	Status();
	
	xResetInterno := FALSE;
	// faz depois dos status o reset automatico do axis
	IF stMotor.Sa.xCmdFwd AND stMotor.Sa.sStatusConexao = 'Parado' AND stHoraAgora.wMilliseconds < 500 THEN
		xResetInterno := TRUE;
	END_IF


END_IF



LeParametros();


xFirstScan := false;

ACTION ControlaACCDEC:

//Pra aparecer na IHM
stMotor.Config.inversor.xtemSuavidadeRampa := TRUE;
stMotor.Config.inversor.xtemACC := TRUE;
stMotor.Config.inversor.xtemDEC := TRUE;

//Pra nao dar exceção
IF stMotor.Config.inversor.SuavidadeRampa < 1 THEN
	stMotor.Config.inversor.SuavidadeRampa := 1;
END_IF
IF stMotor.Config.inversor.SuavidadeRampa > 2 THEN
	stMotor.Config.inversor.SuavidadeRampa := 2;
END_IF

IF stMotor.Config.inversor.ACC < 0.000001 THEN
	stMotor.Config.inversor.ACC := 1;
END_IF

IF stMotor.Config.inversor.DEC < 0.000001 THEN
	stMotor.Config.inversor.DEC := 1;
END_IF

//calculos de verdade
IF xCalcula THEN
	rAux := (stMotor.Sa.iVelocidade*6*stMotor.Config.inversor.SuavidadeRampa)/stMotor.Config.inversor.ACC;
	iAceleracaoCalculada := REAL_TO_UDINT(rAux);
	
	rAux := (stMotor.Sa.iVelocidade*6*stMotor.Config.inversor.SuavidadeRampa)/stMotor.Config.inversor.DEC;
	iDesaceleracaoCalculada := REAL_TO_UDINT(rAux);
	
	rAux := ((stMotor.Sa.iVelocidade*6*stMotor.Config.inversor.SuavidadeRampa)/(stMotor.Config.inversor.ACC*stMotor.Config.inversor.ACC))*((-100.01*stMotor.Config.inversor.SuavidadeRampa)+202.02);
	iJerkCalculado := REAL_TO_UDINT(rAux);
END_IF

//joga nos blocos que precisa
ExAxMvVelo.Acceleration := iAceleracaoCalculada;
ExAxMvVelo.Deceleration := iDesaceleracaoCalculada;
fbMC_Halt.Deceleration := iDesaceleracaoCalculada;


ExAxMvVelo.Jerk := iJerkCalculado;
fbMC_Halt.Jerk := (iJerkCalculado);
ExAxStop.Jerk := (iJerkCalculado);
END_ACTION

ACTION LeParametros:






CASE iEstadoLeCorrente OF
	0: 
		tonEsperaInicio(IN:= TRUE, PT:= T#10S, Q=> , ET=> );
		IF tonEsperaInicio.q THEN
			iEstadoLeCorrente := 1;
		END_IF

	1:

		// tem que no primeiro ciclo jogar uma real nele pra ele conseguir ler depois, nao faz seentido mas vai entender a beckhoffs
		fbReadCorrenteDePico.Execute := TRUE;
		fbReadCorrenteDePico(
			Axis    := AxisREF,
			Idn     := P_0_IDNs + 92,
			Element := 16#40,
			pDstBuf := ADR(rPCorrenteDePico),
			BufLen  := SIZEOF(rPCorrenteDePico),
			Timeout := DEFAULT_ADS_TIMEOUT,
		);
		iEstadoLeCorrente := 2;

		
	2:
		//ai aqui ele so joga um false pra ele nao ficar preso em nada
		fbReadCorrenteDePico(Axis:= AxisREF);
		IF NOT fbReadCorrenteDePico.Busy THEN
			fbReadCorrenteDePico.Execute := FALSE;
			iEstadoLeCorrente := 3;
		END_IF
		
	3:
		//aqui ele faz a logica de verdade e ajeita e fica tudo certo
		IF iAuxCorrenteDePico = 0 AND NOT fbReadCorrenteDePico.Busy THEN
			fbReadCorrenteDePico.Execute := TRUE;
		END_IF
		
		
		fbReadCorrenteDePico(
			Axis    := AxisREF,
			Idn     := P_0_IDNs + 92,
			Element := 16#40,
			pDstBuf := ADR(iAuxCorrenteDePico),
			BufLen  := SIZEOF(iAuxCorrenteDePico),
			Timeout := DEFAULT_ADS_TIMEOUT,
		 );
		
		
		IF NOT fbReadCorrenteDePico.Busy THEN
			fbReadCorrenteDePico.Execute := FALSE;
			fbReadCorrenteDePico(Axis := AxisREF);
			rPCorrenteDePico := iAuxCorrenteDePico;
			rPCorrenteDePico := rPCorrenteDePico/1000;
		END_IF

		
END_CASE
END_ACTION

ACTION Status:


//Erro

ExAxLeErro(
	Axis:= AxisREF, 
	Enable:= TRUE, 
	Valid=> , 
	Busy=> , 
	Error=> , 
	ErrorID=> , 
	AxisErrorID=> );


fbSoEReadDiagNumber(
	Axis:= AxisREF, 
	NetId:= AxisREF.ADS.NetId, 
	Execute:= NOT fbSoEReadDiagNumber.Busy, 
	Timeout:= , 
	Busy=> , 
	Error=> , 
	AdsErrId=> , 
	SercosErrId=> , 
	DiagNumber=> , 
	Attribute=> );
	
fbMCReadStatus(
	Axis:= AxisREF, 
	Enable:= TRUE, 
	Valid=> , 
	Busy=> , 
	Error=> , 
	ErrorID=> , 
	ErrorStop=> , 
	Disabled=> , 
	Stopping=> , 
	StandStill=> , 
	DiscreteMotion=> , 
	ContinuousMotion=> , 
	SynchronizedMotion=> , 
	Homing=> , 
	ConstantVelocity=> , 
	Accelerating=> , 
	Decelerating=> , 
	Status=> );


stMotor.En.xFalhaInversor :=  fbMCReadStatus.Error OR fbSoEReadDiagNumber.DiagNumber < 53266 OR fbSoEReadDiagNumber.DiagNumber > 53268;


fbSoEReadDiagMsg(
	Axis:= AxisREF, 
	NetId:= AxisREF.ADS.NetId, 
	Execute:=  NOT fbSoEReadDiagMsg.Busy, 
	Timeout:= , 
	Busy=> , 
	Error=> , 
	AdsErrId=> , 
	SercosErrId=> , 
	DiagMessage=> , 
	Attribute=> );
	
tonOnline(IN:= fbSoEReadDiagMsg.AdsErrId = 0, PT:= T#5S, Q=> , ET=> );
stMotor.En.xInversorOnline := tonOnline.q;

	
IF fbSoEReadDiagNumber.DiagNumber < 53266 OR fbSoEReadDiagNumber.DiagNumber > 53268 THEN
	stMotor.Sa.sStatusConexao := 'Falha';
	stMotor.Sa.sUltimoErro := fbSoEReadDiagMsg.DiagMessage.strData;
ELSE
	CASE AxisREF.NcToPlc.AxisState OF
		0 :stMotor.Sa.sStatusConexao := 'Parado';
		1,3 :stMotor.Sa.sStatusConexao := 'Rodando';
		4 :stMotor.Sa.sStatusConexao := 'Acelerando';
		5 :stMotor.Sa.sStatusConexao := 'Desacelerando';
	END_CASE
END_IF

IF NOT stMotor.En.xInversorOnline THEN
	stMotor.Sa.sStatusConexao := 'Offline';
END_IF



//Velo
ExAxVeloReal(
	Axis:= AxisREF, 
	Enable:= TRUE, 
	Valid=> , 
	Busy=> , 
	Error=> , 
	ErrorID=> , 
	ActualVelocity=> );
	
IF ExAxVeloReal.ActualVelocity > 1 THEN	
	stMotor.Sa.rVelocidadeRPM := LREAL_TO_REAL(AxisREF.NcToPlc.ActVelo/6);
ELSE
	stMotor.Sa.rVelocidadeRPM := 0;
END_IF


//Temp
(*
ExAxLeTempMotor(
	Axis:= AxisREF, 
	NetId:= '', 
	Execute:= NOT ExAxLeTempMotor.Busy, 
	Timeout:= , 
	Busy=> , 
	Error=> , 
	AdsErrId=> , 
	SercosErrId=> , 
	MotorTemperature=> , 
	Attribute=> );
*)
raux := iTemperaturaMotor;
stMotor.Sa.rTemperaturaMotor := raux/100;//ExAxLeTempMotor.MotorTemperature;

raux := iTemperaturaInversor;
stMotor.Sa.rTemperaturaInver := raux/100;

//Corrente
raux := iCorrente;

iBufferAbsoluteCurrent[iCurrentIndex] := iCorrente;
iCurrentIndex := iCurrentIndex + 1;
IF iCurrentIndex > 10 THEN
	iCurrentIndex := 0;
END_IF
(*
stMotor.Sa.rCorrente := (((iBufferAbsoluteCurrent[0] + 
					iBufferAbsoluteCurrent[1] + iBufferAbsoluteCurrent[2] +
					iBufferAbsoluteCurrent[3] + iBufferAbsoluteCurrent[4] +
					iBufferAbsoluteCurrent[5] + iBufferAbsoluteCurrent[6] +
					iBufferAbsoluteCurrent[7] + iBufferAbsoluteCurrent[8] +
					iBufferAbsoluteCurrent[9])/100)*rPCorrenteDePico)/100;*)
	
				
filtroCorrente(in:= (((raux)/100)*rPCorrenteDePico)/10, T:= T#500MS, K:= 1, out=> stMotor.Sa.rCorrente );		

IF NOT stMotor.Sa.xLigado THEN
	stMotor.Sa.rCorrente := 0;
END_IF

//Torque

stMotor.Sa.rTorque := AxisREF.NcToPlc.ActTorque;

IF NOT stMotor.Sa.xLigado THEN
	stMotor.Sa.rTorque := 0;
END_IF

//Tensao de entrada

stMotor.Sa.rVoltagemEntrada := 0;


stMotor.LeiturasInversorIHM.sCorrente			:= concat(TO_STRING(F_RetiraCasa(stMotor.Sa.rCorrente, 2)), ' A');
stMotor.LeiturasInversorIHM.sStatusConexao		:= stMotor.Sa.sStatusConexao;
stMotor.LeiturasInversorIHM.sTemperaturaInver	:= 'ND';
stMotor.LeiturasInversorIHM.sTemperaturaMotor	:= 'ND';
stMotor.LeiturasInversorIHM.sTorque				:= concat(TO_STRING(F_RetiraCasa(stMotor.Sa.rTorque, 2)), ' %');
stMotor.LeiturasInversorIHM.sUltimoErro			:= stMotor.Sa.sUltimoErro;
//stMotor.LeiturasInversorIHM.sVelocidadeHz		:= concat(TO_STRING(F_RetiraCasa(stMotor.Sa.rVelocidadeRPM, 2)), ' Hz');
stMotor.LeiturasInversorIHM.sVelocidadeRPM		:= concat(TO_STRING(F_RetiraCasa(stMotor.Sa.rVelocidadeRPM, 2)), ' RPM');
END_ACTION

END_FUNCTION_BLOCK

// POUs/Comunicação/CAN/FB_ComunicacaoCanOpen
//{attribute 'hide_all_locals'}
FUNCTION_BLOCK FB_ComunicacaoCanOpen
VAR_IN_OUT
	stMotor	: st_Partida;
	LinkCan	: ATV320_Can;
	Config	: Config_CAN;
END_VAR
VAR_INPUT

END_VAR
VAR_OUTPUT
	ITH_S	: REAL;	//corrente maxima 
	ACC_S	: REAL;	//rampa de aceleração
	DEC_S	: REAL;	//rampa de desaceleração
END_VAR
VAR

	//Maquina
	Ult2ETA	: WORD;
	Ult1ETA	: WORD;

	iEstadoMaquina : MaquinaCanOpen;

	//Escrita SDO
	SDO_WRITE		: ARRAY[1..4] OF SDO_WRITE;
	ReadData		: ARRAY[0..255] OF BYTE;
	WriteDataCTRL	: ARRAY[0..255] OF BYTE;
	uiControlWord	: INT;

	xForcaNST : BOOL;

	//Leitura e escrita
	SDO_READ		: ARRAY[1..4] OF SDO_READ;
	rtComacaLeitura	: R_TRIG;

	ChegouInformacao	: ARRAY[1..4] OF R_TRIG;
	R_TRIGs				: ARRAY[1..10] OF R_TRIG;

	AuxLeitura	: UINT;
	rAux		: REAL;
	
	xAux : BOOL;
	
	iUltimoErro : UINT;
	rtEntrouEmFalha : R_TRIG;
	xPegaUltimoErro : BOOL;
	rtVoltouOnline : R_TRIG;
	
	rtDesligou : R_TRIG;
	iSeguraAlgunsCiclos : INT;

END_VAR


IF xLicensaValida5154156 THEN	
	
	stMotor.En.xTemInversor := TRUE;
	stMotor.En.xResetBlocoComunicacao := FALSE;
	
	Leituras_SDO();
	TrocaEstadoMaquinaDeEstados();
	AcaoMaquinaDeEstados();
	//EscritaPDO();
	Status();
	Escritas_SDO();
	
	// local bloqueado ou em emergencia
	IF xForcaNST OR stMotor.En.xBloqueado (* OR NOT stMotor.En.xEmergenciaOK *) THEN
		LinkCan.Controlword := 0;
	END_IF
ELSE
	ValidaLicensa();
END_IF

ACTION AcaoMaquinaDeEstados:


CASE iEstadoMaquina OF
	SwitchOnDisabled:
		//fica pulsando o sinal para caso ele demore um pouco pra começar a processar os pacotes, ai ele nao fica preso em NST
		IF stMotor.En.stHoraAgora.wMilliseconds > 500 THEN
			LinkCan.Controlword := 16#0006; // manda acionar o drive
		ELSE
			LinkCan.Controlword := 16#0000; // Se comando 
		END_IF

	ReadyToSwitchOn:
		IF stMotor.Sa.xCmdFwd OR stMotor.Sa.xCmdRev THEN
			LinkCan.Controlword := 16#000F; // manda ligar o drive
		END_IF

	SwitchedOn:
		IF stMotor.Sa.xCmdFwd OR stMotor.Sa.xCmdRev THEN
			LinkCan.Controlword := 16#000F; // manda ligar de vez
		ELSE
			LinkCan.Controlword := 16#0007; // manda voltar e e ficar esperando
		END_IF

	OperationEnabled:
		IF NOT (stMotor.Sa.xCmdFwd OR stMotor.Sa.xCmdRev) THEN
			LinkCan.Controlword := 16#0007; // manda desligar o drive
		END_IF

	QuickStopActive:
		LinkCan.Controlword := 16#0000; // a pincipio nao se cai aqui mas caso aconteca ele volta certo

	fault: // caso mandem ele resetar, ou se a falha for COF(erro na can)
		//Caso a falha seja de can ele tenta fazer o reset automatico,
		// ai ele fica pulsando o reset pra caso ele nao pegue o primeiro pacote de reset
		
		LinkCan.Controlword := 16#0006; // manda acionar o drive
		IF (iUltimoErro = 34 AND stMotor.En.xFalhaInversor) THEN
			IF stMotor.En.stHoraAgora.wMilliseconds > 500 THEN
				LinkCan.Controlword := 16#0080; // comando de reset
				stMotor.En.xResetBlocoComunicacao := TRUE;
			ELSE
				LinkCan.Controlword := 16#0000; // Se comando 
			END_IF
		END_IF

		IF stMotor.Sa.xResetParaInversor THEN
			LinkCan.Controlword := 16#0080; // comando de reset
		END_IF

END_CASE

IF stMotor.Sa.xCmdRev THEN
	LinkCan.TargetVelocity := -stMotor.Sa.iVelocidade;
ELSE
	LinkCan.TargetVelocity := stMotor.Sa.iVelocidade;
END_IF

IF stMotor.Sa.xCmdFwd THEN
	IF stMotor.Sa.xResetParaInversor THEN
		LinkCan.TargetVelocity := stMotor.Sa.iVelocidade - 1;
	END_IF
END_IF
END_ACTION

ACTION EscritaPDO:



(*
rtDesligou(CLK:=NOT stMotor.Sa.xLigado);
IF rtDesligou.q OR  iSeguraAlgunsCiclos > 0 AND iSeguraAlgunsCiclos < 20 THEN
	iSeguraAlgunsCiclos := iSeguraAlgunsCiclos +1;
	rAux := Config.Retentiva.NPR-0.1;
	LinkCan.NC1 := REAL_TO_UINT(rAux*10);
	rAux := Config.Retentiva.ITH-0.1;
	LinkCan.NC2 := REAL_TO_UINT(rAux-0.1*10);
	rAux := Config.Retentiva.NSP-0.1;
	LinkCan.NC3 := REAL_TO_UINT(rAux-0.1*10);
	rAux := Config.Retentiva.NCR-0.1;
	LinkCan.NC4 := REAL_TO_UINT(rAux-0.1*10);
ELSE	
	iSeguraAlgunsCiclos := 0;
	LinkCan.NC1 := REAL_TO_UINT(Config.Retentiva.NPR*10);
	LinkCan.NC2 := REAL_TO_UINT(Config.Retentiva.ITH*10);
	LinkCan.NC3 := REAL_TO_UINT(Config.Retentiva.NSP*10);
	LinkCan.NC4 := REAL_TO_UINT(Config.Retentiva.NCR*10);
END_IF
*)
END_ACTION

ACTION Escritas_SDO:

//Corrente
(*
R_TRIGs[1](CLK := Config.normal.xEscreve_ITH, Q =>);

IF R_TRIGs[1].q THEN
	SDO_WRITE[1].StartWriting := TRUE;
END_IF

uiControlWord := TO_INT(Config.Retentiva.ITH_E * 10);
MEMCPY(destAddr := ADR(WriteDataCTRL), srcAddr := ADR(uiControlWord), n := SIZEOF(WriteDataCTRL));

SDO_WRITE[1]
	(
		ADSNetID := Config.Retentiva.sAdressCAN,
			PortNr := 4096 + Config.Retentiva.wPortNrCAN,
			CO_Index := 16#2042,
			CO_SubIndex := 16#17,
			DataLength := SIZEOF(WORD),
			StartWriting :=,
			WriteData := WriteDataCTRL,
			WriteDataFinished =>,
			Error =>);

R_TRIGs[2](CLK := SDO_WRITE[1].WriteDataFinished, Q =>);

IF R_TRIGs[2].q THEN
	Config.normal.xEscreve_ITH	:= FALSE;
	SDO_WRITE[1].StartWriting	:= FALSE;

	Config.normal.xLe := TRUE;
END_IF
*)
//Aceleração

R_TRIGs[3](CLK := Config.normal.xEscreve_ACC, Q =>);

IF R_TRIGs[3].q THEN
	SDO_WRITE[2].StartWriting := TRUE;
END_IF

uiControlWord := TO_INT(Config.Retentiva.ACC_E * 10);
MEMCPY(destAddr := ADR(WriteDataCTRL), srcAddr := ADR(uiControlWord), n := SIZEOF(WriteDataCTRL));

SDO_WRITE[2]
	(
		ADSNetID := Config.Retentiva.sAdressCAN,
			PortNr := 4096 + Config.Retentiva.wPortNrCAN,
			CO_Index := 16#203C,
			CO_SubIndex := 16#2,
			DataLength := SIZEOF(WORD),
			StartWriting :=,
			WriteData := WriteDataCTRL,
			WriteDataFinished =>,
			Error =>);

R_TRIGs[4](CLK := SDO_WRITE[2].WriteDataFinished, Q =>);

IF R_TRIGs[4].q THEN
	SDO_WRITE[2].StartWriting	:= FALSE;
	Config.normal.xEscreve_ACC	:= FALSE;

	Config.normal.xLe := TRUE;
END_IF

//Desaceleração

R_TRIGs[5](CLK := Config.normal.xEscreve_DEC, Q =>);

IF R_TRIGs[5].q THEN
	SDO_WRITE[3].StartWriting := TRUE;
END_IF

uiControlWord := TO_INT(Config.Retentiva.DEC_E * 10);
MEMCPY(destAddr := ADR(WriteDataCTRL), srcAddr := ADR(uiControlWord), n := SIZEOF(WriteDataCTRL));

SDO_WRITE[3]
	(
		ADSNetID := Config.Retentiva.sAdressCAN,
			PortNr := 4096 + Config.Retentiva.wPortNrCAN,
			CO_Index := 16#203C,
			CO_SubIndex := 16#3,
			DataLength := SIZEOF(WORD),
			StartWriting :=,
			WriteData := WriteDataCTRL,
			WriteDataFinished =>,
			Error =>);

R_TRIGs[6](CLK := SDO_WRITE[3].WriteDataFinished, Q =>);

IF R_TRIGs[6].q THEN
	SDO_WRITE[3].StartWriting	:= FALSE;
	Config.normal.xEscreve_DEC	:= FALSE;

	Config.normal.xLe := true;
END_IF
END_ACTION

ACTION Leituras_SDO:

rtComacaLeitura(CLK := Config.Normal.xLe, Q =>);

IF rtComacaLeitura.Q THEN
	//xTerminouLeituras:=FALSE;
END_IF
(*
//////////// ITH
SDO_READ[1]
	(
		StartReading :=,
			CO_Index := 16#2042,
			CO_SubIndex := 16#17,
			DataLength := SIZEOF(UINT),
			PortNr := 4096 + Config.Retentiva.wPortNrCAN,
			ADSNetID := Config.Retentiva.sAdressCAN);

ChegouInformacao[1](CLK := SDO_READ[1].ReadDataAvailable, Q =>);

IF ChegouInformacao[1].q THEN
	Config.Normal.xLe			:= FALSE;
	SDO_READ[2].StartReading	:= TRUE;

	ReadData := SDO_READ[1].ReadData;
	MEMCPY(destAddr := ADR(AuxLeitura), srcAddr := ADR(ReadData), n := SIZEOF(UINT));
	ITH_S					:= UINT_TO_REAL(AuxLeitura) / 10;
	Config.Retentiva.ITH_E	:= ITH_S;
END_IF
*)
//////////// ACC		
SDO_READ[2]
	(
		StartReading := Config.Normal.xLe,
			CO_Index := 16#203C,
			CO_SubIndex := 16#2,
			DataLength := SIZEOF(UINT),
			PortNr := 4096 + Config.Retentiva.wPortNrCAN,
			ADSNetID := Config.Retentiva.sAdressCAN);

ChegouInformacao[2](CLK := SDO_READ[2].ReadDataAvailable, Q =>);

IF ChegouInformacao[2].q THEN
	SDO_READ[2].StartReading	:= FALSE;
	SDO_READ[3].StartReading	:= TRUE;

	ReadData := SDO_READ[2].ReadData;
	MEMCPY(destAddr := ADR(AuxLeitura), srcAddr := ADR(ReadData), n := SIZEOF(UINT));
	ACC_S					:= UINT_TO_REAL(AuxLeitura) / 10;
	Config.Retentiva.ACC_E	:= ACC_S;
END_IF

//////////// DEC		
SDO_READ[3]
	(
		StartReading :=,
			CO_Index := 16#203C,
			CO_SubIndex := 16#3,
			DataLength := SIZEOF(UINT),
			PortNr := 4096 + Config.Retentiva.wPortNrCAN,
			ADSNetID := Config.Retentiva.sAdressCAN);

ChegouInformacao[3](CLK := SDO_READ[3].ReadDataAvailable, Q =>);

IF ChegouInformacao[3].q THEN
	SDO_READ[3].StartReading := FALSE;

	ReadData := SDO_READ[3].ReadData;
	MEMCPY(destAddr := ADR(AuxLeitura), srcAddr := ADR(ReadData), n := SIZEOF(UINT));
	DEC_S					:= UINT_TO_REAL(AuxLeitura) / 10;
	Config.Retentiva.DEC_E	:= DEC_S;
END_IF




SDO_READ[4]
	(
		StartReading :=xPegaUltimoErro,
			CO_Index := 16#2029,
			CO_SubIndex := 16#16,
			DataLength := SIZEOF(UINT),
			PortNr := 4096 + Config.Retentiva.wPortNrCAN,
			ADSNetID := Config.Retentiva.sAdressCAN);

ChegouInformacao[4](CLK := SDO_READ[4].ReadDataAvailable, Q =>);

IF ChegouInformacao[4].q THEN
	xPegaUltimoErro := FALSE;
	ReadData := SDO_READ[4].ReadData;
	MEMCPY(destAddr := ADR(iUltimoErro), srcAddr := ADR(ReadData), n := SIZEOF(UINT));
END_IF
END_ACTION

ACTION Status:

// manda status de online e falha
stMotor.En.xFalhaInversor := iEstadoMaquina = Fault;

//IF  THEN
	IF LinkCan.NodeState <> 31 THEN
		stMotor.En.xInversorOnline :=
			 (LinkCan.NodeState <> 2); // Nao sei se é o melhor jeito, mas o 2 é o unico que fala especificamente de o inversor nao ter sido encontrado
										// nao o 31 pq se nao ele buga e fica dando reset pra sempre nos inversor	
	END_IF
//END_IF
								
rAux							:= LinkCan.NM2;
stMotor.Sa.rCorrente			:= rAux / 10;
stMotor.Sa.rTemperaturaMotor	:= LinkCan.NM3;
rAux							:= LinkCan.NM4;
stMotor.Sa.rTorque				:= rAux/10;

stMotor.Sa.rVelocidadeRPM	:= LinkCan.ControlEffort;
rAux						:= stMotor.Sa.rVelocidadeRPM;
stMotor.Sa.rVelocidadeHZ	:= rAux * 0.016667 * 2;

stMotor.LeiturasInversorIHM.sCorrente			:= concat(TO_STRING(F_RetiraCasa(stMotor.Sa.rCorrente, 2)), ' A');
stMotor.LeiturasInversorIHM.sStatusConexao		:= stMotor.Sa.sStatusConexao;
stMotor.LeiturasInversorIHM.sTemperaturaInver	:= 'ND';
stMotor.LeiturasInversorIHM.sTemperaturaMotor	:= concat(TO_STRING(F_RetiraCasa(stMotor.Sa.rTemperaturaMotor, 2)), ' %');
stMotor.LeiturasInversorIHM.sTorque				:= concat(TO_STRING(F_RetiraCasa(stMotor.Sa.rTorque, 2)), ' %');
stMotor.LeiturasInversorIHM.sUltimoErro			:= stMotor.Sa.sUltimoErro;
stMotor.LeiturasInversorIHM.sVelocidadeHz		:= concat(TO_STRING(F_RetiraCasa(stMotor.Sa.rVelocidadeHZ, 2)), ' Hz');

IF stMotor.Config.xVeloEmMetroPMin THEN
	rAux										:= (stMotor.Sa.rVelocidadeRPM * stMotor.Config.rVeloEmMetroPMin_Conversao) / 1800;	
	stMotor.Sa.rVeloComissionada				:= rAux;
	stMotor.LeiturasInversorIHM.sVelocidadeRPM	:= concat(TO_STRING(F_RetiraCasa(rAux, 2)), ' m/Min');
ELSIF stMotor.Config.xVeloEmPorcentagem THEN
	IF stMotor.Config.rVeloEmPorcentagem_VeloMax < 0.1 THEN
		stMotor.Config.rVeloEmPorcentagem_VeloMax := 1;
	END_IF
	rAux										:= (stMotor.Sa.rVelocidadeRPM * 100) / stMotor.Config.rVeloEmPorcentagem_VeloMax;
	stMotor.Sa.rVeloComissionada				:= rAux;
	stMotor.LeiturasInversorIHM.sVelocidadeRPM	:= concat(TO_STRING(F_RetiraCasa(rAux, 2)), ' %');
ELSE
	stMotor.Sa.rVeloComissionada				:= stMotor.Sa.rVelocidadeRPM;
	stMotor.LeiturasInversorIHM.sVelocidadeRPM := concat(TO_STRING(F_RetiraCasa(stMotor.Sa.rVelocidadeRPM, 2)), ' RPM');
END_IF

stMotor.LeiturasInversorIHM.sVoltagemEntrada := 'ND';

config.Normal.rITH_Lido	:= ITH_S;
config.Normal.rACC_Lido	:= ACC_S;
config.Normal.rDEC_Lido	:= DEC_S;

// 30 é STO
xAux := LinkCan.NM1 = 30;
stMotor.En.xEmergenciaOK := stMotor.En.xEmergenciaOK AND NOT xAux;

CASE LinkCan.NM1 OF
	0:
		IF iUltimoErro = 0 THEN
			stMotor.Sa.sStatusConexao := 'Offline';
		ELSE
			stMotor.Sa.sStatusConexao := '[Autotuning] (TUN)';
		END_IF

	1:
		stMotor.Sa.sStatusConexao := '[Injeção de CC] (DCB)';

	2:
		stMotor.Sa.sStatusConexao := '[Pronto] (RDY)';

	3:
		stMotor.Sa.sStatusConexao := '[Esperando] (NST)';

	4:
		stMotor.Sa.sStatusConexao := '[Rodando] (RUN)';

	5:
		stMotor.Sa.sStatusConexao := '[Acelerando] (ACC)';

	6:
		stMotor.Sa.sStatusConexao := '[Desacelerando] (DEC)';

	7:
		stMotor.Sa.sStatusConexao := '[Limitando Corrente] (CLI)';

	8:
		stMotor.Sa.sStatusConexao := '[Parada Rapida] (FST)';

	11:
		stMotor.Sa.sStatusConexao := '[Sem Tensão de Entrada] (NLP)';

	13:
		stMotor.Sa.sStatusConexao := '[control.stop] (CTL)';

	14:
		stMotor.Sa.sStatusConexao := '[Dec. adapt.] (OBR)';

	15:
		stMotor.Sa.sStatusConexao := '[Output cut] (SOC)';

	17:
		stMotor.Sa.sStatusConexao := '[Undervoltage Warning] (USA)';

	18:
		stMotor.Sa.sStatusConexao := '[TC Mode Active] (TC)';

	19:
		stMotor.Sa.sStatusConexao := '[In autotest] (ST)';

	20:
		stMotor.Sa.sStatusConexao := '[Autotest error] (FA)';

	21:
		stMotor.Sa.sStatusConexao := '[Autotest OK] (OK)';

	22:
		stMotor.Sa.sStatusConexao := '[EEprom test] (EP))';

	23:
		stMotor.Sa.sStatusConexao := '[Falha] (FLT)';

	25:
		stMotor.Sa.sStatusConexao := '[DCP Flashing Mode] (DCP)';

	30:
		stMotor.Sa.sStatusConexao := '[Emergencia Ativa] (STO)';

	35:
		stMotor.Sa.sStatusConexao := '[Salvando Energia] (IDLE)';

	36:
		stMotor.Sa.sStatusConexao := '[Atualizando Firmware] (FWUP)';

	37:
		stMotor.Sa.sStatusConexao := '[AFE Mains Undervoltage ] (URA)';
END_CASE

IF NOT stMotor.En.xInversorOnline THEN
	stMotor.Sa.sStatusConexao := 'Offline';
END_IF

CASE iUltimoErro OF
	0:
		stMotor.Sa.sUltimoErro := 'Carregando';

	2:
		stMotor.Sa.sUltimoErro := '[EEPROM Control] (EEF1)';

	3:
		stMotor.Sa.sUltimoErro := '[Configuração Incorreta] (CFF)';

	4:
		stMotor.Sa.sUltimoErro := '[Configuração Invalida] (CFI)';

	5:
		stMotor.Sa.sUltimoErro := '[Com. ModBus Interrompida] (SLF1)';

	6:
		stMotor.Sa.sUltimoErro := '[Internal Link Error] (ILF)';

	7:
		stMotor.Sa.sUltimoErro := '[Fieldbus Com Interrupt] (CNF)';

	8:
		stMotor.Sa.sUltimoErro := '[Erro Externo] (EPF1)';

	9:
		stMotor.Sa.sUltimoErro := '[Sobrecorrente] (OCF)';

	10:
		stMotor.Sa.sUltimoErro := '[Precharge Capacitor] (CRF1)';

	11:
		stMotor.Sa.sUltimoErro := '[Encoder Feedback Loss] (SPF)';

	12:
		stMotor.Sa.sUltimoErro := '[Load slipping] (ANF)';

	15:
		stMotor.Sa.sUltimoErro := '[Entrada Superaquecendo] (IHF)';

	16:
		stMotor.Sa.sUltimoErro := '[Inversor Superaquecendo] (OHF)';

	17:
		stMotor.Sa.sUltimoErro := '[Motor Sobracarregado] (OLF)';

	18:
		stMotor.Sa.sUltimoErro := '[DC Bus Sobretensão] (OBF)';

	19:
		stMotor.Sa.sUltimoErro := '[Entrada com Sobretensão] (OSF)';

	20:
		stMotor.Sa.sUltimoErro := '[Perda de 1 Fase da Saida] (OPF1)';

	21:
		stMotor.Sa.sUltimoErro := '[Perda de Fase na Entrada] (PHF)';

	22:
		stMotor.Sa.sUltimoErro := '[Entrada em subtensão] (USF)';

	23:
		stMotor.Sa.sUltimoErro := '[Motor em Curto-Circuito] (SCF1)';

	24:
		stMotor.Sa.sUltimoErro := '[Motor Overspeed] (SOF)';

	25:
		stMotor.Sa.sUltimoErro := '[Autotuning Error] (TNF)';

	26:
		stMotor.Sa.sUltimoErro := '[Internal Error 1] (INF1)';

	27:
		stMotor.Sa.sUltimoErro := '[Internal Error 2] (INF2)';

	28:
		stMotor.Sa.sUltimoErro := '[Internal Error 3] (INF3)';

	29:
		stMotor.Sa.sUltimoErro := '[Internal Error 4] (INF4)';

	30:
		stMotor.Sa.sUltimoErro := '[EEPROM Power] (EEF2)';

	32:
		stMotor.Sa.sUltimoErro := '[Curto-Circuito a Terra] (SCF3)';

	33:
		stMotor.Sa.sUltimoErro := '[Falta de Fase na Saida] (OPF2)';

	34:
		stMotor.Sa.sUltimoErro := '[Com. CANopen Interrompida] (COF)';

	35:
		stMotor.Sa.sUltimoErro := '[Brake Control] (BLF)';

	37:
		stMotor.Sa.sUltimoErro := '[Internal Error 7] (INF7)';

	38:
		stMotor.Sa.sUltimoErro := '[Fieldbus Error] (EPF2)';

	40:
		stMotor.Sa.sUltimoErro := '[Internal Error 8] (INF8)';

	41:
		stMotor.Sa.sUltimoErro := '[Brake Feedback] (BRF)';

	42:
		stMotor.Sa.sUltimoErro := '[PC Com. Interruption] (SLF2)';

	43:
		stMotor.Sa.sUltimoErro := '[Encoder Coupling] (ECF)';

	44:
		stMotor.Sa.sUltimoErro := '[Erro na Limitção de Torque] (SSF)';

	45:
		stMotor.Sa.sUltimoErro := '[Com. HMI Interrompido] (SLF3)';

	51:
		stMotor.Sa.sUltimoErro := '[Internal Error 9] (INF9)';

	52:
		stMotor.Sa.sUltimoErro := '[Internal Error 10] (INFA)';

	53:
		stMotor.Sa.sUltimoErro := '[Internal Error 11] (INFB)';

	54:
		stMotor.Sa.sUltimoErro := '[IGBT Superaquecendo] (TJF)';

	55:
		stMotor.Sa.sUltimoErro := '[IGBT em Curto-Circuito] (SCF4)';

	56:
		stMotor.Sa.sUltimoErro := '[Motor em Curto-Circuito] (SCF5)';

	57:
		stMotor.Sa.sUltimoErro := '[Torque timeout] (SRF)';

	58:
		stMotor.Sa.sUltimoErro := '[Out Contact Closed Error] (FCF1)';

	59:
		stMotor.Sa.sUltimoErro := '[Out Contact Opened Error] (FCF2)';

	60:
		stMotor.Sa.sUltimoErro := '[Internal Error 12] (INFC)';

	62:
		stMotor.Sa.sUltimoErro := '[Encoder] (ENF)';

	64:
		stMotor.Sa.sUltimoErro := '[Input Contactor] (LCF)';

	65:
		stMotor.Sa.sUltimoErro := '[DB unit sh. circuit] (BUF)';

	68:
		stMotor.Sa.sUltimoErro := '[Internal Error 6] (INF6)';

	69:
		stMotor.Sa.sUltimoErro := '[Internal Error 14] (INFE)';

	70:
		stMotor.Sa.sUltimoErro := '[Braking Resistor ovld] (BOF)';

	71:
		stMotor.Sa.sUltimoErro := '[Perda AI3 4-20mA] (LFF3)';

	72:
		stMotor.Sa.sUltimoErro := '[Perda AI4 4-20mA] (LFF4)';

	73:
		stMotor.Sa.sUltimoErro := '[Boards Compatibility] (HCF)';

	76:
		stMotor.Sa.sUltimoErro := '[Dynamic Load Error] (DLF)';

	77:
		stMotor.Sa.sUltimoErro := '[Conf Transfer Error] (CFI2)';

	79:
		stMotor.Sa.sUltimoErro := '[Perda AI5 4-20 mA] (LFF5)';

	99:
		stMotor.Sa.sUltimoErro := '[Channel Switch Error] (CSF)';

	100:
		stMotor.Sa.sUltimoErro := '[Process Underload] (ULF)';

	101:
		stMotor.Sa.sUltimoErro := '[Process Overload] (OLC)';

	105:
		stMotor.Sa.sUltimoErro := '[Angle error] (ASF)';

	106:
		stMotor.Sa.sUltimoErro := '[Perda AI1 4-20 mA] (LFF1)';

	107:
		stMotor.Sa.sUltimoErro := '[Safety Function Error] (SAFF)';

	112:
		stMotor.Sa.sUltimoErro := '[AI3 Th Level Error] (TH3F)';

	113:
		stMotor.Sa.sUltimoErro := '[AI3 Thermal Sensor Error] (T3CF)';

	120:
		stMotor.Sa.sUltimoErro := '[AI4 Th Level Error] (TH4F)';

	121:
		stMotor.Sa.sUltimoErro := '[AI4 Thermal Sensor Error] (T4CF)';

	122:
		stMotor.Sa.sUltimoErro := '[AI5 Th Level Error] (TH5F)';

	123:
		stMotor.Sa.sUltimoErro := '[AI5 Thermal Sensor Error] (T5CF)';

	128:
		stMotor.Sa.sUltimoErro := '[Program Loading Error] (PGLF)';

	129:
		stMotor.Sa.sUltimoErro := '[Program Running Error] (PGRF)';

	142:
		stMotor.Sa.sUltimoErro := '[Internal Error 16] (INFG)';

	143:
		stMotor.Sa.sUltimoErro := '[Internal Error 17] (INFH)';

	144:
		stMotor.Sa.sUltimoErro := '[Internal Error 0] (INF0)';

	146:
		stMotor.Sa.sUltimoErro := '[Internal Error 13] (INFD)';

	148:
		stMotor.Sa.sUltimoErro := '[Motor Stall Error] (STF)';

	149:
		stMotor.Sa.sUltimoErro := '[Internal Error 21] (INFL)';

	150:
		stMotor.Sa.sUltimoErro := '[Com. Embd Eth Interrompida] (ETHF)';

	151:
		stMotor.Sa.sUltimoErro := '[Internal Error 15] (INFF)';

	152:
		stMotor.Sa.sUltimoErro := '[Firmware Update Error] (FWER)';

	153:
		stMotor.Sa.sUltimoErro := '[Internal Error 22] (INFM)';

	154:
		stMotor.Sa.sUltimoErro := '[Internal Error 25] (INFP)';

	155:
		stMotor.Sa.sUltimoErro := '[Internal Error 20] (INFK)';

	156:
		stMotor.Sa.sUltimoErro := '[Internal Error 19] (INFJ)';

	157:
		stMotor.Sa.sUltimoErro := '[Internal Error 27] (INFR)';

	158:
		stMotor.Sa.sUltimoErro := '[Internal Error 23] (INFN)';

	159:
		stMotor.Sa.sUltimoErro := '[AFE ShortCircuit error] (SCF6)';

	160:
		stMotor.Sa.sUltimoErro := '[AFE Bus unbalancing ] (OBF2)';

	161:
		stMotor.Sa.sUltimoErro := '[Internal Error 28] (INFS)';

	173:
		stMotor.Sa.sUltimoErro := '[Cabinet Overheat  Error] (CHF)';

	175:
		stMotor.Sa.sUltimoErro := '[Internal Error 31] (INFV)';

	176:
		stMotor.Sa.sUltimoErro := '[Internal Error 29] (INFT)';

	177:
		stMotor.Sa.sUltimoErro := '[Internal Error 30] (INFU)';

	179:
		stMotor.Sa.sUltimoErro := '[AFE IGBT over-heat error] (TJF2)';

	180:
		stMotor.Sa.sUltimoErro := '[AFE contactor feedback error] (CRF3)';

	181:
		stMotor.Sa.sUltimoErro := '[Pre-settings Transfer Error] (CFI3)';

	182:
		stMotor.Sa.sUltimoErro := '[Circuit Breaker Error] (CBF)';

	184:
		stMotor.Sa.sUltimoErro := '[DB unit op. circuit] (BUFO)';

	185:
		stMotor.Sa.sUltimoErro := '[Inversor Sobrecarregado] (TLOF)';

	186:
		stMotor.Sa.sUltimoErro := '[MultiDrive Link Error] (MDLF)';

	187:
		stMotor.Sa.sUltimoErro := '[AI1 Th Level Error] (TH1F)';

	188:
		stMotor.Sa.sUltimoErro := '[AI1 Thermal Sensor Error] (T1CF)';

	189:
		stMotor.Sa.sUltimoErro := '[Backlash Error] (BSQF)';

	190:
		stMotor.Sa.sUltimoErro := '[M/S Device Error] (MSDF)';

	194:
		stMotor.Sa.sUltimoErro := '[Encoder Th Level Error] (THEF)';

	195:
		stMotor.Sa.sUltimoErro := '[Encoder Th Sensor Error] (TECF)';

	196:
		stMotor.Sa.sUltimoErro := '[Sem Configuração] (CFI4)';

	200:
		stMotor.Sa.sUltimoErro := '[FDR 1 Error] (FDR1)';

	201:
		stMotor.Sa.sUltimoErro := '[FDR 2 Error] (FDR2)';

	206:
		stMotor.Sa.sUltimoErro := '[DC Bus Ripple Error] (DCRE)';

	208:
		stMotor.Sa.sUltimoErro := '[Egy Saving Exit Error] (IDLF)';

	209:
		stMotor.Sa.sUltimoErro := '[Load Mvt Error] (MDCF)';
END_CASE
END_ACTION

ACTION TrocaEstadoMaquinaDeEstados:

Ult2ETA	:= LinkCan.StatusWord AND 16#00FF;
Ult1ETA	:= LinkCan.StatusWord AND 16#000F;

CASE Ult2ETA OF
	16#0040:
		iEstadoMaquina := SwitchOnDisabled;

	16#0050:
		iEstadoMaquina := SwitchOnDisabled;

	16#0021:
		iEstadoMaquina := ReadyToSwitchOn;

	16#0031:
		iEstadoMaquina := ReadyToSwitchOn;

	16#0033:
		iEstadoMaquina := SwitchedOn;

	16#0037:
		iEstadoMaquina := OperationEnabled;

	16#0017:
		iEstadoMaquina := QuickStopActive;
END_CASE

//Independendte do estado quando estiver assim é pq ta em erro
// pela palavra que vem na rede ou por ele estar offline
//So deixa mandar o reset se ele estiver em falha
IF Ult1ETA = 16#0008 THEN
	iEstadoMaquina := Fault;
END_IF


rtEntrouEmFalha(CLK := iEstadoMaquina = Fault);
rtVoltouOnline(CLK := stMotor.En.xInversorOnline);
IF rtEntrouEmFalha.q OR rtVoltouOnline.q THEN
	xPegaUltimoErro := TRUE;
	iUltimoErro := 0;
END_IF
END_ACTION

END_FUNCTION_BLOCK

// POUs/Comunicação/Ethernet/ConversaoBilateralConfig
FUNCTION_BLOCK ConversaoBilateralConfig
VAR_IN_OUT
	Base		: UINT;
	Convertida	: REAL;
END_VAR
VAR_INPUT
	multiplicador : INT := 10;
END_VAR
VAR_OUTPUT
END_VAR
VAR
	rAuxConversao				: REAL;
	rUltimaVariavelConvertida	: REAL;
	rUltimaVariavelBase			: REAL;
END_VAR

IF xLicensaValida5154156 THEN
	
	IF Convertida <> rUltimaVariavelConvertida THEN
		Base := TO_UINT(Convertida * multiplicador);
	END_IF
	
	IF Base <> rUltimaVariavelBase THEN
		rAuxConversao	:= Base;
		Convertida		:= (rAuxConversao / multiplicador);
	END_IF
	
	rUltimaVariavelConvertida	:= Convertida;
	rUltimaVariavelBase			:= Base;

ELSE
	ValidaLicensa();	
END_IF

END_FUNCTION_BLOCK

// POUs/Comunicação/Ethernet/FB_ComunicacaoEthernet
FUNCTION_BLOCK FB_ComunicacaoEthernet
VAR_IN_OUT
	stMotor	: st_Partida;
	Config	: ConfigComunicacaoEthernet;
END_VAR
VAR_OUTPUT
	rLSP				: REAL;	//velocidade minima
	rHSP				: REAL;	//velocidade maxima
	rTRF				: REAL;	//maxima velocidade
	rITH				: REAL;	//corrente maxima 
	rACC				: REAL;	//rampa de aceleração
	rDEC				: REAL;	//rampa de desaceleração
	xPHR				: BOOL;	//ordem das fases
	xEscreveParametros	: BOOL;
	xLerParametros		: BOOL;
	sIPAdress			: STRING(15); //Endereço Ethernet do Inversor
END_VAR
VAR

	RegistradoresEscrita	: ARRAY[1..2] OF st_ReadWriteREG;
	RegisWrite				: ARRAY[1..2] OF FB_MBWriteSingleReg;

	RegistradoresLeitura	: ARRAY[1..11] OF st_ReadWriteREG;
	RegisRead				: ARRAY[1..11] OF FB_MBReadRegs;

	RegistradoresAmbos	: ARRAY[1..7] OF st_ReadWriteREG;
	RegisAmbosRead		: ARRAY[1..7] OF FB_MBReadRegs;
	RegisAmbosWrite		: ARRAY[1..7] OF FB_MBWriteSingleReg;
	fbControleBilateral	: ARRAY[1..7] OF ConversaoBilateralConfig;

	//escrita
	CMD		: WORD;	//Palavra de comando
	LFRD	: INT;	//Velocidade de comando

	//leitura
	ETA		: WORD;	//palavra de status
	HMIS	: WORD;	//status da IHM
	LFT		: WORD;	//ultimo erro
	RFRD	: INT;	//velo agora
	RFR		: INT;	// velo em HZ
	OTR		: INT;	//Torque Motor
	THR		: UINT;	//Temp Motor
	LCR		: UINT;	//Corrente Motor
	ULN		: UINT;	//voltagem na entrada
	THD		: UINT;	//temperatura inversor
	APPS	: WORD;	//Local remoto

	//Ambos
	LSP					: UINT;	//velocidade minima
	HSP					: UINT;	//velocidade maxima
	TRF					: UINT;	//maxima velocidade
	ITH					: UINT;	//corrente maxima 
	ACC					: UINT;	//rampa de aceleração
	DEC					: UINT;	//rampa de desaceleração
	PHR					: UINT;	//ordem das fases
	rtComacaLer			: R_TRIG;
	rtComacaEscrever	: R_TRIG;
	ftTerminou			: ARRAY[1..22] OF F_TRIG;
	xConfigOk			: BOOL;
	rAuxPHR				: REAL;
	rAuxPHR2			: REAL;

	//Maquina de estados
	iStatusWordHexa		: INT;
	byteStatusWord		: BYTE;
	strHexStatusWord	: STRING;
	iMachineState		: INT;
	bWriteReg			: BOOL;
	iEstadoMaquina : MaquinaCanOpen;
	Ult2ETA	: WORD;
	Ult1ETA	: WORD;

	//xOnline
	tonOnline	: TON;
	rUltimaULN	: UINT;

	//Outros
	sAux			: STRING;
	xCiclo1s		: BOOL;
	xCiclo01s		: BOOL;
	ton1			: TON;
	ton01			: TON;
	I				: INT;
	J				: INT	:= 1;
	PrimeiroScan	: BOOL	:= TRUE;
	rAuxs			: REAL;
	xAux			: BOOL;
END_VAR

IF xLicensaValida5154156 THEN
	
//========================================================================
//FB de comunicação Ethernet com ATV da TEKNIKE
//feito por Tiago Bortolini Cunico em 18/09/2021
//foi usado codigo feito pelo Ricardo Gajardo tambem
//Este bloco foi criado especificamente para ser utilizado jusntamente com
//o bloco da partida sendo necessario somente linkar o st_motor igual ao da
//partida e o config para os parametros do motor
//========================================================================
	
	Ciclo1s();
	Leituras();
	Leituras_Escritas();
	
	TrocaEstadoMaquinaDeEstados();
	AcaoMaquinaDeEstados();
	
	Escrita();
	
	IHM();
	
	sIPAdress			:= Config.sIPAdress;
	xEscreveParametros	:= Config.xEscreveParametros;
	xLerParametros		:= Config.xLerParametros;
	
	stMotor.En.xTemInversor := TRUE;
	
	PrimeiroScan	:= FALSE;
	I				:= J;
ELSE
	ValidaLicensa();
END_IF

ACTION AcaoMaquinaDeEstados:

CASE iEstadoMaquina OF
	SwitchOnDisabled:
		//fica pulsando o sinal para caso ele demore um pouco pra começar a processar os pacotes, ai ele nao fica preso em NST
		IF stMotor.En.stHoraAgora.wMilliseconds > 500 THEN
			CMD := 16#0006; // manda acionar o drive
		ELSE
			CMD := 16#0000; // Se comando 
		END_IF

	ReadyToSwitchOn:
		IF stMotor.Sa.xCmdFwd OR stMotor.Sa.xCmdRev THEN
			CMD := 16#000F; // manda ligar o drive
		END_IF

	SwitchedOn:
		IF stMotor.Sa.xCmdFwd OR stMotor.Sa.xCmdRev THEN
			CMD := 16#000F; // manda ligar de vez
		ELSE
			CMD := 16#0007; // manda voltar e e ficar esperando
		END_IF

	OperationEnabled:
		IF NOT (stMotor.Sa.xCmdFwd OR stMotor.Sa.xCmdRev) THEN
			CMD := 16#0007; // manda desligar o drive
		END_IF

	QuickStopActive:
		CMD := 16#0000; // a pincipio nao se cai aqui mas caso aconteca ele volta certo

	fault: // caso mandem ele resetar, ou se a falha for COF(erro na can)
		//Caso a falha seja de can ele tenta fazer o reset automatico,
		// ai ele fica pulsando o reset pra caso ele nao pegue o primeiro pacote de reset
		
		IF stMotor.Sa.xResetParaInversor THEN
			CMD := 16#0080; // comando de reset
		ELSE
			CMD := 16#0000; // Se comando 
		END_IF
		
		IF (LFT = 150 AND stMotor.En.xFalhaInversor) THEN
			IF stMotor.En.stHoraAgora.wMilliseconds > 500 THEN
				CMD := 16#0080; // comando de reset
			ELSE
				CMD := 16#0000; // Se comando 
			END_IF
		END_IF
		

		

END_CASE



IF stMotor.Sa.xCmdRev THEN
	LFRD := -stMotor.Sa.iVelocidade;
ELSE
	LFRD := stMotor.Sa.iVelocidade;
END_IF

IF stMotor.Sa.xCmdFwd THEN
	IF stMotor.Sa.xResetParaInversor THEN
		LFRD := stMotor.Sa.iVelocidade - 1;
	END_IF
END_IF
END_ACTION

ACTION Ciclo1s:

ton1.IN := TRUE;

IF ton1.q THEN
	ton1.IN		:= FALSE;
	xCiclo1s	:= NOT xCiclo1s;
END_IF

ton1(IN :=, PT := T#0.250S, Q =>, ET =>);

ton01.IN := TRUE;

IF ton01.q THEN
	ton01.IN	:= FALSE;
	xCiclo01s	:= NOT xCiclo01s;
END_IF

ton01(IN :=, PT := T#0.1S, Q =>, ET =>);
END_ACTION

ACTION Escrita:

IF PrimeiroScan THEN
	RegistradoresEscrita[1].nMBAddr	:= 8501;
	RegistradoresEscrita[2].nMBAddr	:= 8602;
END_IF

RegistradoresEscrita[1].nValue		:= (CMD);
RegistradoresEscrita[1].xEscreve	:= xCiclo01s;

//LFRD								:= stMotor.Sa.iVelocidade;
//Velocidade definida na maquina de estado
RegistradoresEscrita[2].nValue		:= TO_WORD(LFRD);
RegistradoresEscrita[2].xEscreve	:= xCiclo01s;

FOR I := 1 TO 2 DO
	RegistradoresEscrita[i].nQuantity := 1;

	RegisWrite[i]
		(
			sIPAddr := Config.sIPAdress,
				nTCPPort := 502,
				nUnitID := 0,
				nMBAddr := RegistradoresEscrita[i].nMBAddr,
				nValue := RegistradoresEscrita[i].nValue,
				bExecute := RegistradoresEscrita[i].xEscreve,
				tTimeout := T#1S,
				bBusy => RegistradoresEscrita[i].bBusy,
				bError => RegistradoresEscrita[i].bError,
				nErrId => RegistradoresEscrita[i].nErrId);

END_FOR
END_ACTION

ACTION IHM:

stMotor.LeiturasInversorIHM.sCorrente			:= TO_STRING(F_RetiraCasa(stMotor.Sa.rCorrente, 2));
stMotor.LeiturasInversorIHM.sStatusConexao		:= stMotor.Sa.sStatusConexao;
stMotor.LeiturasInversorIHM.sTemperaturaInver	:= TO_STRING(F_RetiraCasa(stMotor.Sa.rTemperaturaInver, 2));
stMotor.LeiturasInversorIHM.sTemperaturaMotor	:= TO_STRING(F_RetiraCasa(stMotor.Sa.rTemperaturaMotor, 2));
stMotor.LeiturasInversorIHM.sTorque				:= TO_STRING(F_RetiraCasa(stMotor.Sa.rTorque, 2));
stMotor.LeiturasInversorIHM.sUltimoErro			:= stMotor.Sa.sUltimoErro;
stMotor.LeiturasInversorIHM.sVelocidadeHz		:= TO_STRING(F_RetiraCasa(stMotor.Sa.rVelocidadeHz, 2));
stMotor.LeiturasInversorIHM.sVelocidadeRPM		:= TO_STRING(F_RetiraCasa(stMotor.Sa.rVelocidadeRPM, 2));
stMotor.LeiturasInversorIHM.sVoltagemEntrada	:= TO_STRING(F_RetiraCasa(stMotor.Sa.rVoltagemEntrada, 2));
END_ACTION

ACTION Leituras:

IF PrimeiroScan THEN
	RegistradoresLeitura[1].nMBAddr		:= 3201;
	RegistradoresLeitura[1].cbLength	:= SIZEOF(ETA);
	RegistradoresLeitura[1].pDestAddr	:= ADR(ETA);

	RegistradoresLeitura[2].nMBAddr		:= 3240;
	RegistradoresLeitura[2].cbLength	:= SIZEOF(HMIS);
	RegistradoresLeitura[2].pDestAddr	:= ADR(HMIS);

	RegistradoresLeitura[3].nMBAddr		:= 7121;
	RegistradoresLeitura[3].cbLength	:= SIZEOF(LFT);
	RegistradoresLeitura[3].pDestAddr	:= ADR(LFT);

	RegistradoresLeitura[4].nMBAddr		:= 8604;
	RegistradoresLeitura[4].cbLength	:= SIZEOF(RFRD);
	RegistradoresLeitura[4].pDestAddr	:= ADR(RFRD);

	RegistradoresLeitura[5].nMBAddr		:= 3205;
	RegistradoresLeitura[5].cbLength	:= SIZEOF(OTR);
	RegistradoresLeitura[5].pDestAddr	:= ADR(OTR);

	RegistradoresLeitura[6].nMBAddr		:= 9630;
	RegistradoresLeitura[6].cbLength	:= SIZEOF(THR);
	RegistradoresLeitura[6].pDestAddr	:= ADR(THR);

	RegistradoresLeitura[7].nMBAddr		:= 3204;
	RegistradoresLeitura[7].cbLength	:= SIZEOF(LCR);
	RegistradoresLeitura[7].pDestAddr	:= ADR(LCR);

	RegistradoresLeitura[8].nMBAddr		:= 3207;
	RegistradoresLeitura[8].cbLength	:= SIZEOF(ULN);
	RegistradoresLeitura[8].pDestAddr	:= ADR(ULN);

	RegistradoresLeitura[9].nMBAddr		:= 3209;
	RegistradoresLeitura[9].cbLength	:= SIZEOF(THD);
	RegistradoresLeitura[9].pDestAddr	:= ADR(THD);

	RegistradoresLeitura[10].nMBAddr	:= 15980;
	RegistradoresLeitura[10].cbLength	:= SIZEOF(APPS);
	RegistradoresLeitura[10].pDestAddr	:= ADR(APPS);

	RegistradoresLeitura[11].nMBAddr	:= 3202;
	RegistradoresLeitura[11].cbLength	:= SIZEOF(RFR);
	RegistradoresLeitura[11].pDestAddr	:= ADR(RFR);
END_IF

FOR I := 1 TO 11 DO
	RegistradoresLeitura[I].nQuantity	:= 1;
	RegistradoresLeitura[I].xLe			:= xCiclo1s;

	RegisRead[i]
		(
			sIPAddr := Config.sIPAdress,
				nTCPPort := 502,
				nUnitID := 0,
				nQuantity := RegistradoresLeitura[I].nQuantity,
				nMBAddr := RegistradoresLeitura[I].nMBAddr,
				cbLength := RegistradoresLeitura[I].cbLength,
				pDestAddr := RegistradoresLeitura[I].pDestAddr,
				bExecute := RegistradoresLeitura[I].xLe,
				tTimeout := T#1S,
				bBusy => RegistradoresLeitura[I].bBusy,
				bError => RegistradoresLeitura[I].bError,
				nErrId => RegistradoresLeitura[I].nErrID,
				cbRead => RegistradoresLeitura[I].cbRead);
END_FOR

//Tratamento dos dados
rAuxs							:= LCR;
stMotor.Sa.rCorrente			:= rAuxs / 100;
rAuxs							:= THD;
stMotor.Sa.rTemperaturaInver	:= rAuxs;
rAuxs							:= THR;
stMotor.Sa.rTemperaturaMotor	:= rAuxs;
rAuxs							:= OTR;
stMotor.Sa.rTorque				:= rAuxs / 10;
rAuxs							:= RFR;
stMotor.Sa.rVelocidadeHz		:= rAuxs / 10;
rAuxs							:= RFRD;
stMotor.Sa.rVelocidadeRPM		:= rAuxs;
rAuxs							:= ULN;
stMotor.Sa.rVoltagemEntrada		:= rAuxs / 10;

//Controle se ele ta online
tonOnline(IN:= RegistradoresLeitura[1].bError OR RegistradoresLeitura[1].bBusy, PT:=T#5S , Q=> , ET=> );
stMotor.En.xInversorOnline	:= NOT tonOnline.q;

//Se ele ta em falha
stMotor.En.xFalhaInversor	:= HMIS = 23;
//se ele ta em emergencia
stMotor.En.xEmergenciaOK 	:= HMIS <> 30;
//Se esta em local ou remoto
stMotor.En.xLocal 			:= APPS = 2;
stMotor.En.xTemInversor		:= TRUE;

CASE HMIS OF
	0:
		stMotor.Sa.sStatusConexao := '[Autotuning] (TUN)';

	1:
		stMotor.Sa.sStatusConexao := '[Injeção de CC] (DCB)';

	2:
		stMotor.Sa.sStatusConexao := '[Pronto] (RDY)';

	3:
		stMotor.Sa.sStatusConexao := '[Roda livre] (NST)';

	4:
		stMotor.Sa.sStatusConexao := '[Rodando] (RUN)';

	5:
		stMotor.Sa.sStatusConexao := '[Acelerando] (ACC)';

	6:
		stMotor.Sa.sStatusConexao := '[Desacelerando] (DEC)';

	7:
		stMotor.Sa.sStatusConexao := '[Limitação de corrente] (CLI)';

	8:
		stMotor.Sa.sStatusConexao := '[Parada rapida] (FST)';

	11:
		stMotor.Sa.sStatusConexao := '[Sem tensão na entrada] (NLP)';

	13:
		stMotor.Sa.sStatusConexao := '[Controle de parada] (CTL)';

	14:
		stMotor.Sa.sStatusConexao := '[Desaceleração adaptativa] (OBR)';

	15:
		stMotor.Sa.sStatusConexao := '[Output cut] (SOC)';

	17:
		stMotor.Sa.sStatusConexao := '[Alerta de subtansão] (USA)';

	18:
		stMotor.Sa.sStatusConexao := '[TC Mode Active] (TC)';

	19:
		stMotor.Sa.sStatusConexao := '[Em autoteste] (ST)';

	20:
		stMotor.Sa.sStatusConexao := '[Autoteste erro] (FA)';

	21:
		stMotor.Sa.sStatusConexao := '[Autoteste OK] (OK)';

	22:
		stMotor.Sa.sStatusConexao := '[EEprom test] (EP))';

	23:
		stMotor.Sa.sStatusConexao := '[Falha] (FLT)';

	25:
		stMotor.Sa.sStatusConexao := '[DCP Flashing Mode] (DCP)';

	30:
		stMotor.Sa.sStatusConexao := '[Emergencia ativa] (STO)';

	35:
		stMotor.Sa.sStatusConexao := '[Energy Saving] (IDLE)';

	36:
		stMotor.Sa.sStatusConexao := '[Firmware Update] (FWUP)';

	37:
		stMotor.Sa.sStatusConexao := '[AFE Mains Undervoltage ] (URA)';
END_CASE

CASE LFT OF
	0:
		stMotor.Sa.sUltimoErro := '[No Error] (NOF)';

	2:
		stMotor.Sa.sUltimoErro := '[EEPROM Control] (EEF1)';

	3:
		stMotor.Sa.sUltimoErro := '[Configuração incorreta] (CFF)';

	4:
		stMotor.Sa.sUltimoErro := '[Configuração invalida] (CFI)';

	5:
		stMotor.Sa.sUltimoErro := '[Erro na comunicação modbus] (SLF1)';

	6:
		stMotor.Sa.sUltimoErro := '[Internal Link Error] (ILF)';

	7:
		stMotor.Sa.sUltimoErro := '[Fieldbus Com Interrupt] (CNF)';

	8:
		stMotor.Sa.sUltimoErro := '[Erro externo] (EPF1)';

	9:
		stMotor.Sa.sUltimoErro := '[Sobrecorrente] (OCF)';

	10:
		stMotor.Sa.sUltimoErro := '[Precarregando capacitor] (CRF1)';

	11:
		stMotor.Sa.sUltimoErro := '[Encoder Feedback Loss] (SPF)';

	12:
		stMotor.Sa.sUltimoErro := '[Carga escorregando] (ANF)';

	15:
		stMotor.Sa.sUltimoErro := '[Entrada sobreaquecendo] (IHF)';

	16:
		stMotor.Sa.sUltimoErro := '[Inversor sobreaquecendo] (OHF)';

	17:
		stMotor.Sa.sUltimoErro := '[Motor sobrecarregado] (OLF)';

	18:
		stMotor.Sa.sUltimoErro := '[DC Bus sobretensão] (OBF)';

	19:
		stMotor.Sa.sUltimoErro := '[Bobretensão na entrada] (OSF)';

	20:
		stMotor.Sa.sUltimoErro := '[Perda de 1 fase de saida] (OPF1)';

	21:
		stMotor.Sa.sUltimoErro := '[Perda de fase na entrada] (PHF)';

	22:
		stMotor.Sa.sUltimoErro := '[Subtensão na entrada] (USF)';

	23:
		stMotor.Sa.sUltimoErro := '[Motor em curto] (SCF1)';

	24:
		stMotor.Sa.sUltimoErro := '[Motor em sobrevelocidade] (SOF)';

	25:
		stMotor.Sa.sUltimoErro := '[Autotuning Error] (TNF)';

	26:
		stMotor.Sa.sUltimoErro := '[Internal Error 1] (INF1)';

	27:
		stMotor.Sa.sUltimoErro := '[Internal Error 2] (INF2)';

	28:
		stMotor.Sa.sUltimoErro := '[Internal Error 3] (INF3)';

	29:
		stMotor.Sa.sUltimoErro := '[Internal Error 4] (INF4)';

	30:
		stMotor.Sa.sUltimoErro := '[EEPROM Power] (EEF2)';

	32:
		stMotor.Sa.sUltimoErro := '[Curto a terra] (SCF3)';

	33:
		stMotor.Sa.sUltimoErro := '[Perda das fases da saida] (OPF2)';

	34:
		stMotor.Sa.sUltimoErro := '[CanOpen error] (COF)';

	35:
		stMotor.Sa.sUltimoErro := '[Brake Control] (BLF)';

	37:
		stMotor.Sa.sUltimoErro := '[Internal Error 7] (INF7)';

	38:
		stMotor.Sa.sUltimoErro := '[Fieldbus Error] (EPF2)';

	40:
		stMotor.Sa.sUltimoErro := '[Internal Error 8] (INF8)';

	41:
		stMotor.Sa.sUltimoErro := '[Brake Feedback] (BRF)';

	42:
		stMotor.Sa.sUltimoErro := '[Comunicação com o PC interrompida] (SLF2)';

	43:
		stMotor.Sa.sUltimoErro := '[Encoder Coupling] (ECF)';

	44:
		stMotor.Sa.sUltimoErro := '[Erro na limitação de torque] (SSF)';

	45:
		stMotor.Sa.sUltimoErro := '[Perda de comunicação com a IHM] (SLF3)';

	51:
		stMotor.Sa.sUltimoErro := '[Internal Error 9] (INF9)';

	52:
		stMotor.Sa.sUltimoErro := '[Internal Error 10] (INFA)';

	53:
		stMotor.Sa.sUltimoErro := '[Internal Error 11] (INFB)';

	54:
		stMotor.Sa.sUltimoErro := '[IGBT sobreaquecendo] (TJF)';

	55:
		stMotor.Sa.sUltimoErro := '[IGBT em curto] (SCF4)';

	56:
		stMotor.Sa.sUltimoErro := '[Motor em curto] (SCF5)';

	57:
		stMotor.Sa.sUltimoErro := '[Torque timeout] (SRF)';

	58:
		stMotor.Sa.sUltimoErro := '[Out Contact Closed Error] (FCF1)';

	59:
		stMotor.Sa.sUltimoErro := '[Out Contact Opened Error] (FCF2)';

	60:
		stMotor.Sa.sUltimoErro := '[Internal Error 12] (INFC)';

	62:
		stMotor.Sa.sUltimoErro := '[Encoder] (ENF)';

	64:
		stMotor.Sa.sUltimoErro := '[Input Contactor] (LCF)';

	65:
		stMotor.Sa.sUltimoErro := '[DB unit sh. circuit] (BUF)';

	68:
		stMotor.Sa.sUltimoErro := '[Internal Error 6] (INF6)';

	69:
		stMotor.Sa.sUltimoErro := '[Internal Error 14] (INFE)';

	70:
		stMotor.Sa.sUltimoErro := '[Braking Resistor ovld] (BOF)';

	71:
		stMotor.Sa.sUltimoErro := '[AI3 4-20mA loss] (LFF3)';

	72:
		stMotor.Sa.sUltimoErro := '[AI4 4-20mA loss] (LFF4)';

	73:
		stMotor.Sa.sUltimoErro := '[Boards Compatibility] (HCF)';

	76:
		stMotor.Sa.sUltimoErro := '[Dynamic Load Error] (DLF)';

	77:
		stMotor.Sa.sUltimoErro := '[Conf Transfer Error] (CFI2)';

	79:
		stMotor.Sa.sUltimoErro := '[AI5 4-20 mA loss] (LFF5)';

	99:
		stMotor.Sa.sUltimoErro := '[Channel Switch Error] (CSF)';

	100:
		stMotor.Sa.sUltimoErro := '[Process Underload] (ULF)';

	101:
		stMotor.Sa.sUltimoErro := '[Process Overload] (OLC)';

	105:
		stMotor.Sa.sUltimoErro := '[Angle error] (ASF)';

	106:
		stMotor.Sa.sUltimoErro := '[AI1 4-20 mA loss] (LFF1)';

	107:
		stMotor.Sa.sUltimoErro := '[Safety Function Error] (SAFF)';

	112:
		stMotor.Sa.sUltimoErro := '[AI3 Th Level Error] (TH3F)';

	113:
		stMotor.Sa.sUltimoErro := '[AI3 Thermal Sensor Error] (T3CF)';

	120:
		stMotor.Sa.sUltimoErro := '[AI4 Th Level Error] (TH4F)';

	121:
		stMotor.Sa.sUltimoErro := '[AI4 Thermal Sensor Error] (T4CF)';

	122:
		stMotor.Sa.sUltimoErro := '[AI5 Th Level Error] (TH5F)';

	123:
		stMotor.Sa.sUltimoErro := '[AI5 Thermal Sensor Error] (T5CF)';

	128:
		stMotor.Sa.sUltimoErro := '[Program Loading Error] (PGLF)';

	129:
		stMotor.Sa.sUltimoErro := '[Program Running Error] (PGRF)';

	142:
		stMotor.Sa.sUltimoErro := '[Internal Error 16] (INFG)';

	143:
		stMotor.Sa.sUltimoErro := '[Internal Error 17] (INFH)';

	144:
		stMotor.Sa.sUltimoErro := '[Internal Error 0] (INF0)';

	146:
		stMotor.Sa.sUltimoErro := '[Internal Error 13] (INFD)';

	148:
		stMotor.Sa.sUltimoErro := '[Motor Stall Error] (STF)';

	149:
		stMotor.Sa.sUltimoErro := '[Internal Error 21] (INFL)';

	150:
		stMotor.Sa.sUltimoErro := '[Ethernet error] (ETHF)';

	151:
		stMotor.Sa.sUltimoErro := '[Internal Error 15] (INFF)';

	152:
		stMotor.Sa.sUltimoErro := '[Firmware Update Error] (FWER)';

	153:
		stMotor.Sa.sUltimoErro := '[Internal Error 22] (INFM)';

	154:
		stMotor.Sa.sUltimoErro := '[Internal Error 25] (INFP)';

	155:
		stMotor.Sa.sUltimoErro := '[Internal Error 20] (INFK)';

	156:
		stMotor.Sa.sUltimoErro := '[Internal Error 19] (INFJ)';

	157:
		stMotor.Sa.sUltimoErro := '[Internal Error 27] (INFR)';

	158:
		stMotor.Sa.sUltimoErro := '[Internal Error 23] (INFN)';

	159:
		stMotor.Sa.sUltimoErro := '[AFE ShortCircuit error] (SCF6)';

	160:
		stMotor.Sa.sUltimoErro := '[AFE Bus unbalancing ] (OBF2)';

	161:
		stMotor.Sa.sUltimoErro := '[Internal Error 28] (INFS)';

	173:
		stMotor.Sa.sUltimoErro := '[Cabinet Overheat  Error] (CHF)';

	175:
		stMotor.Sa.sUltimoErro := '[Internal Error 31] (INFV)';

	176:
		stMotor.Sa.sUltimoErro := '[Internal Error 29] (INFT)';

	177:
		stMotor.Sa.sUltimoErro := '[Internal Error 30] (INFU)';

	179:
		stMotor.Sa.sUltimoErro := '[AFE IGBT over-heat error] (TJF2)';

	180:
		stMotor.Sa.sUltimoErro := '[AFE contactor feedback error] (CRF3)';

	181:
		stMotor.Sa.sUltimoErro := '[Pre-settings Transfer Error] (CFI3)';

	182:
		stMotor.Sa.sUltimoErro := '[Circuit Breaker Error] (CBF)';

	184:
		stMotor.Sa.sUltimoErro := '[DB unit op. circuit] (BUFO)';

	185:
		stMotor.Sa.sUltimoErro := '[Inversor sobrecarregado] (TLOF)';

	186:
		stMotor.Sa.sUltimoErro := '[MultiDrive Link Error] (MDLF)';

	187:
		stMotor.Sa.sUltimoErro := '[AI1 Th Level Error] (TH1F)';

	188:
		stMotor.Sa.sUltimoErro := '[AI1 Thermal Sensor Error] (T1CF)';

	189:
		stMotor.Sa.sUltimoErro := '[Backlash Error] (BSQF)';

	190:
		stMotor.Sa.sUltimoErro := '[M/S Device Error] (MSDF)';

	194:
		stMotor.Sa.sUltimoErro := '[Encoder Th Level Error] (THEF)';

	195:
		stMotor.Sa.sUltimoErro := '[Encoder Th Sensor Error] (TECF)';

	196:
		stMotor.Sa.sUltimoErro := '[Empty Configuration] (CFI4)';

	200:
		stMotor.Sa.sUltimoErro := '[FDR 1 Error] (FDR1)';

	201:
		stMotor.Sa.sUltimoErro := '[FDR 2 Error] (FDR2)';

	206:
		stMotor.Sa.sUltimoErro := '[DC Bus Ripple Error] (DCRE)';

	208:
		stMotor.Sa.sUltimoErro := '[Egy Saving Exit Error] (IDLF)';

	209:
		stMotor.Sa.sUltimoErro := '[Load Mvt Error] (MDCF)';
END_CASE

CASE WORD_TO_INT(APPS) OF
	0:
		sAux := 'Rodando';

	1:
		sAux := 'Parado';

	2:
		sAux := ' Oper. Local';

	3:
		sAux := 'Oper. Ethernet';

	4:
		sAux := 'Modo manual';

	5:
		sAux := 'PID Ativo';

	6:
		sAux := 'Anti-Jam In progress';

	7:
		sAux := 'Flow limit In progress';

	8:
		sAux := 'PipeFill In progress';

	9:
		sAux := 'Jockey Pump Active';

	10:
		sAux := 'Boost In progress';

	11:
		sAux := 'Sleep Active';

	12:
		sAux := 'Priming Pump Active';

	13:
		sAux := 'InletPres Comp In progress';
END_CASE

IF sAux = ' Oper. Local' THEN
	stMotor.Sa.sStatusConexao := CONCAT(stMotor.Sa.sStatusConexao, sAux);
END_IF
END_ACTION

ACTION Leituras_Escritas:

IF PrimeiroScan THEN
	RegistradoresAmbos[1].nMBAddr	:= 3105;
	RegistradoresAmbos[1].cbLength	:= SIZEOF(LSP);
	RegistradoresAmbos[1].pDestAddr	:= ADR(LSP);

	RegistradoresAmbos[2].nMBAddr	:= 3104;
	RegistradoresAmbos[2].cbLength	:= SIZEOF(HSP);
	RegistradoresAmbos[2].pDestAddr	:= ADR(HSP);

	RegistradoresAmbos[3].nMBAddr	:= 3103;
	RegistradoresAmbos[3].cbLength	:= SIZEOF(TRF);
	RegistradoresAmbos[3].pDestAddr	:= ADR(TRF);

	RegistradoresAmbos[4].nMBAddr	:= 9622;
	RegistradoresAmbos[4].cbLength	:= SIZEOF(ITH);
	RegistradoresAmbos[4].pDestAddr	:= ADR(ITH);

	RegistradoresAmbos[5].nMBAddr	:= 9001;
	RegistradoresAmbos[5].cbLength	:= SIZEOF(ACC);
	RegistradoresAmbos[5].pDestAddr	:= ADR(ACC);

	RegistradoresAmbos[6].nMBAddr	:= 9002;
	RegistradoresAmbos[6].cbLength	:= SIZEOF(DEC);
	RegistradoresAmbos[6].pDestAddr	:= ADR(DEC);

	RegistradoresAmbos[7].nMBAddr	:= 13401;
	RegistradoresAmbos[7].cbLength	:= SIZEOF(PHR);
	RegistradoresAmbos[7].pDestAddr	:= ADR(PHR);
END_IF

RegistradoresAmbos[1].nValue	:= TO_UINT(LSP);	//:= TO_UINT(rLSP*10);
RegistradoresAmbos[2].nValue	:= TO_UINT(HSP);	//:= TO_UINT(rHSP*10);
RegistradoresAmbos[3].nValue	:= TO_UINT(TRF);	//:= TO_UINT(rTRF*10);
RegistradoresAmbos[4].nValue	:= TO_UINT(ITH);	//:= TO_UINT(rITH*10);
RegistradoresAmbos[5].nValue	:= TO_UINT(ACC);	//:= TO_UINT(rACC*10);
RegistradoresAmbos[6].nValue	:= TO_UINT(DEC);	//:= TO_UINT(rDEC*10);
RegistradoresAmbos[7].nValue	:= TO_UINT(PHR);	//:= TO_WORD(xPHR);

xConfigOk := LSP < HSP AND HSP > 0 AND HSP <= TRF AND ITH > 0;

rtComacaLer(CLK := Config.xLerParametros, Q =>);

IF rtComacaLer.q THEN
	FOR I := 1 TO 7 DO // so aceita um por vez e quando nao ta ligado
		RegistradoresAmbos[I].xLe := Config.xLerParametros AND NOT Config.xEscreveParametros AND APPS = 1;
	END_FOR
END_IF

rtComacaEscrever(CLK := Config.xEscreveParametros, Q =>);

IF rtComacaEscrever.q THEN
	FOR I := 1 TO 7 DO
		RegistradoresAmbos[I].xEscreve := NOT Config.xLerParametros AND Config.xEscreveParametros AND APPS = 1 AND xConfigOk;
	END_FOR
END_IF

FOR I := 1 TO 7 DO

	RegistradoresAmbos[I].nQuantity := 1;

	RegisAmbosRead[i]
		(
			sIPAddr := Config.sIPAdress,
				nTCPPort := 502,
				nUnitID := 0,
				nQuantity := RegistradoresAmbos[I].nQuantity,
				nMBAddr := RegistradoresAmbos[I].nMBAddr,
				cbLength := RegistradoresAmbos[I].cbLength,
				pDestAddr := RegistradoresAmbos[I].pDestAddr,
				bExecute := RegistradoresAmbos[I].xLe,
				tTimeout := T#1S,
				bBusy => RegistradoresAmbos[I].bBusy,
				bError => RegistradoresAmbos[I].bError,
				nErrId => RegistradoresAmbos[I].nErrID,
				cbRead => RegistradoresAmbos[I].cbRead);

	ftTerminou[i](CLK := RegistradoresAmbos[I].bBusy, Q =>);

	IF ftTerminou[i].q THEN
		RegistradoresAmbos[I].xLe := FALSE;
	END_IF

	RegisAmbosWrite[i]
		(
			sIPAddr := Config.sIPAdress,
				nTCPPort := 502,
				nUnitID := 0,
				nMBAddr := RegistradoresAmbos[i].nMBAddr,
				nValue := RegistradoresAmbos[i].nValue,
				bExecute := RegistradoresAmbos[i].xEscreve,
				tTimeout := T#1S,
				bBusy => RegistradoresAmbos[i].bBusy,
				bError => RegistradoresAmbos[i].bError,
				nErrId => RegistradoresAmbos[i].nErrId);

	ftTerminou[i + 11](CLK := RegistradoresAmbos[I].bBusy, Q =>);

	IF ftTerminou[i + 11].q THEN
		RegistradoresAmbos[I].xEscreve := FALSE;
	END_IF

END_FOR

xAux := FALSE;

FOR I := 1 TO 7 DO
	xAux := xAux OR RegistradoresAmbos[I].xLe;
END_FOR

IF NOT xAux THEN
	Config.xLerParametros := FALSE;
END_IF

xAux := FALSE;

FOR I := 1 TO 7 DO
	xAux := xAux OR RegistradoresAmbos[I].xEscreve;
END_FOR

IF NOT xAux THEN
	Config.xEscreveParametros := FALSE;
END_IF

// para a informação de ida e volta ser na mesma variavel
fbControleBilateral[1](Base := LSP, Convertida := Config.rLSP);
fbControleBilateral[2](Base := HSP, Convertida := Config.rHSP);
fbControleBilateral[3](Base := TRF, Convertida := Config.rTRF);
fbControleBilateral[4](Base := ITH, Convertida := Config.rITH, multiplicador := 100);
fbControleBilateral[5](Base := ACC, Convertida := Config.rACC);
fbControleBilateral[6](Base := DEC, Convertida := Config.rDEC);

// por ser bool nao deu no fb bilateral
IF Config.xPHR <> TO_BOOL(rAuxPHR) THEN
	PHR := TO_UINT(Config.xPHR);
END_IF

IF PHR <> rAuxPHR2 THEN
	Config.xPHR := TO_BOOL(PHR);
END_IF

rAuxPHR		:= TO_REAL(Config.xPHR);
rAuxPHR2	:= PHR;

// joga as variaveis na saida pra aparecer
rLSP	:= Config.rLSP;
rHSP	:= Config.rHSP;
rTRF	:= Config.rTRF;
rITH	:= Config.rITH;
rACC	:= Config.rACC;
rDEC	:= Config.rDEC;
xPHR	:= Config.xPHR;
END_ACTION

ACTION MaquinaDeEstados:

(*Converte valor da Status Word para Hexa*)
byteStatusWord		:= UINT_TO_BYTE(ETA);
strHexStatusWord	:= BYTE_TO_HEXSTR(in := byteStatusWord, iPrecision := 2, bLoCase := FALSE);
iStatusWordHexa		:= STRING_TO_INT(strHexStatusWord);
//iStsWordHexa := iStatusWordHexa;
(*---FIM---*)

IF iStatusWordHexa = 17 AND NOT INT_TO_UINT(iMachineState) = (4) THEN //535
	CMD			:= 0;
	bWriteReg	:= TRUE;

	IF iStatusWordHexa = 50 THEN
		bWriteReg := FALSE;
	END_IF
END_IF

CASE iMachineState OF

	0:															//NST
		IF iStatusWordHexa = 50 OR iStatusWordHexa = 40 THEN	//592
			CMD			:= 6;									//Com o inversor em NST, joga o inversor para 'RDY'
			bWriteReg	:= TRUE;
		END_IF

		IF iStatusWordHexa = 31 OR iStatusWordHexa = 21 THEN //561
			bWriteReg		:= FALSE;
			iMachineState	:= 1; //com o inveror em RDY joga para o passo de ativação do comando
		END_IF

		IF iStatusWordHexa = 33 THEN //563 ou 591
			bWriteReg		:= FALSE;
			iMachineState	:= 2; //com o inveror em RDY e ativado joga para o passo de comando
		END_IF

	1:						//RDY
		CMD			:= 7;	//Com o inversor em RDY, Ativa o Comando
		bWriteReg	:= TRUE;

		IF iStatusWordHexa = 33 THEN //563 ou 591
			bWriteReg		:= FALSE;
			iMachineState	:= 2; //com o inveror em RDY e ativado joga para o passo de comando
		END_IF

		IF iStatusWordHexa = 50 THEN
			iMachineState := 0;
		END_IF

	2: //

		IF iStatusWordHexa = 50 THEN
			iMachineState := 0;
		END_IF

		IF CMD = 15 AND iStatusWordHexa = 33 AND NOT stMotor.Sa.xCmdFwd THEN
			iMachineState := 1;
		END_IF

		IF stMotor.Sa.xCmdFwd THEN
			CMD			:= 15; //Comando de marcha avanço
			bWriteReg	:= TRUE;

			IF iStatusWordHexa = 37 THEN
				bWriteReg		:= FALSE;
				iMachineState	:= 3;
			END_IF
		END_IF

	(*
		IF stMotor.Sa.xCmdRwd THEN 
				CMD:= 2063; //Comando de marcha avanço
				bWriteReg := TRUE;		
			IF iStatusWordHexa=37 THEN
				bWriteReg := FALSE;				
				iMachineState:=5;
			END_IF	
		END_IF	
		*)

	3:
		IF iStatusWordHexa = 37 THEN //1591

			IF NOT stMotor.Sa.xCmdFwd THEN
				CMD			:= 7; //Comando de parada por rampa
				bWriteReg	:= TRUE;
			END_IF

			IF iStatusWordHexa = 33 THEN
				bWriteReg := FALSE;
			END_IF
		END_IF

		(*
			IF NOT stMotor.Sa.xCmdFwd THEN
				
				IF TRUE(*xTipodeParada*) THEN // no momento fica assim 17/09/2021
					
					CMD:= 7; //Comando de parada por rampa
					bWriteReg := TRUE;
					
					IF 	iStatusWordHexa=33 THEN
						bWriteReg := FALSE;
					END_IF	
				ELSE
				
					CMD:= 6; //Comando de parada por inércia
					bWriteReg := TRUE;	
		
					IF 	iStatusWordHexa=31 THEN
						bWriteReg := FALSE;
					END_IF	
			END_IF
		END_IF
				
			IF TRUE (*xParadaRapida*) THEN
				iMachineState:=4;		
			END_IF
		END_IF
		*)

		IF iStatusWordHexa = 31 THEN	//561
			iMachineState := 1;			//com o inveror em RDY joga para o passo de ativação do comando
		END_IF

		IF iStatusWordHexa = 33 THEN	//563
			iMachineState := 2;			//com o inveror em RDY joga para o passo de ativação do comando
		END_IF

		IF iStatusWordHexa = 50 THEN //592
			iMachineState := 6;
		END_IF

	4:
		CMD			:= 2; //Comando de parada rápida		
		bWriteReg	:= TRUE;

		IF iStatusWordHexa = 17 OR iStatusWordHexa = 50 THEN //535
			bWriteReg		:= FALSE;
			iMachineState	:= 0;
		END_IF

	5:
		IF iStatusWordHexa = 37 THEN //34359

			(*
				IF NOT stMotor.Sa.xCmdRwd THEN
					IF xTipodeParada THEN
					CMD:= 7; //Comando de parada por rampa
					bWriteReg := TRUE;
				IF iStatusWordHexa=33 THEN
					bWriteReg := FALSE;
				END_IF			
					ELSE
					CMD:= 6; //Comando de parada por inércia
						bWriteReg := TRUE;
				IF iStatusWordHexa=31 THEN
					bWriteReg := FALSE;
				END_IF			
		
					END_IF
				END_IF
				*)

			IF TRUE THEN //xParadaRapida THEN
				iMachineState := 4;
			END_IF
		END_IF

		IF iStatusWordHexa = 31 THEN	//561
			iMachineState := 1;			//com o inveror em RDY joga para o passo de ativação do comando
		END_IF

		IF iStatusWordHexa = 33 THEN	//563
			iMachineState := 2;			//com o inveror em RDY joga para o passo de ativação do comando
		END_IF

		IF iStatusWordHexa = 50 THEN //592
			iMachineState := 6;
		END_IF

	6:
		CMD			:= 0;
		bWriteReg	:= TRUE;

		IF iStatusWordHexa = 50 THEN
			bWriteReg		:= FALSE;
			iMachineState	:= 0;
		END_IF

	ELSE

		CMD			:= 0; //Comando de parada rápida	
		bWriteReg	:= TRUE;

		IF iStatusWordHexa = 50 THEN
			bWriteReg := FALSE;
		END_IF

END_CASE

IF stMotor.Sa.xResetParaInversor THEN
	CMD			:= 128; //Comando de reset via rede	
	bWriteReg	:= TRUE;

	IF iStatusWordHexa = 50 THEN
		bWriteReg := FALSE;
	END_IF

END_IF

(*Alterei aqui em 22/01*)
IF iStatusWordHexa = 50 THEN
	IF stMotor.Sa.xResetParaInversor THEN
		CMD			:= 128; //Comando de reset via rede	
		bWriteReg	:= TRUE;

		IF iStatusWordHexa = 31 THEN
			bWriteReg := FALSE;
		END_IF
	END_IF
END_IF

(*
	
ELSE
	CMD:= 0;
	bWriteReg := TRUE;
	IF 	iStatusWordHexa= 50 THEN
		bWriteReg := FALSE;
	END_IF		


END_IF
*)
END_ACTION

ACTION TrocaEstadoMaquinaDeEstados:

Ult2ETA	:= ETA AND 16#006F;
Ult1ETA	:= ETA AND 16#000F;

CASE Ult2ETA OF
	16#0040:
		iEstadoMaquina := SwitchOnDisabled;

	16#0021:
		iEstadoMaquina := ReadyToSwitchOn;

	16#0031:
		iEstadoMaquina := ReadyToSwitchOn;

	16#0023:
		iEstadoMaquina := SwitchedOn;

	16#0027:
		iEstadoMaquina := OperationEnabled;

	16#0007:
		iEstadoMaquina := QuickStopActive;
END_CASE

//Independendte do estado quando estiver assim é pq ta em erro
// pela palavra que vem na rede ou por ele estar offline
//So deixa mandar o reset se ele estiver em falha
IF Ult1ETA = 16#0008 THEN
	iEstadoMaquina := Fault;
END_IF
END_ACTION

END_FUNCTION_BLOCK

// POUs/Comunicação/EthernetIP/Delta/FB_DeltaMS
FUNCTION_BLOCK FB_DeltaMS
VAR_IN_OUT
	motor : st_Partida;
	LinkDelta : st_LinkDeltaEIP;
END_VAR
VAR_INPUT
END_VAR
VAR_OUTPUT
END_VAR
VAR
	rAux : REAL;
	rtVoltouEmergencia : R_TRIG;
	i1ParteStatus : INT;
	i2ParteStatus : INT;
	tonOnline : ton;
	tonParaDriverPraTrocarDeReferencia : ton;
END_VAR

Emergencia();

ControleMarcha();
ControleVelocidade();

Status();

Others();

ACTION ControleMarcha:


//Controle Basico de liga e desliga
IF motor.Sa.xLigado THEN
	LinkDelta.Control := 1;
	IF motor.Sa.xCmdFwd THEN
		LinkDelta.Control := 2#010010; //32;
	END_IF
	IF motor.Sa.xCmdRev THEN
		LinkDelta.Control := 2#100010;// 50;
	END_IF
ELSE
	LinkDelta.Control := 1;
END_IF
END_ACTION

ACTION ControleVelocidade:


rAux := motor.Sa.iVelocidade;
rAux := rAux * 0.016666 * 2;

LinkDelta.oFrequenceCommand := REAL_TO_UINT(rAux * 100);
END_ACTION

ACTION Emergencia:




motor.En.xEmergenciaOK := motor.En.xEmergenciaOK AND LinkDelta.ErrorCode <> 76;
END_ACTION

ACTION Others:






//Manda o reset
rtVoltouEmergencia(CLK:= motor.En.xEmergenciaOK, Q=> );
IF rtVoltouEmergencia.q THEN
	motor.en.xResetBlocoComunicacao := TRUE;
END_IF

LinkDelta.Others := 0;

IF motor.Sa.xResetParaInversor OR (motor.En.stHoraAgora.wMilliseconds>500 AND ( NOT motor.En.xEmergenciaOK OR LinkDelta.ErrorCode = 49)) THEN
	LinkDelta.Others := LinkDelta.Others OR 2#010;
ELSE
	LinkDelta.Others := LinkDelta.Others AND 2#101;
END_IF

//Se der emergencia ele ta External Fault (Esse é pra incluir as emergencias por software)
IF NOT motor.En.xEmergenciaOK AND LinkDelta.ErrorCode <> 76 THEN
	LinkDelta.Others := LinkDelta.Others OR 2#001;
ELSE
	LinkDelta.Others := LinkDelta.Others AND 2#110;
END_IF

//Quando bloqueado ele joga um base block, que eu acho que é tipo um NST
IF motor.En.xBloqueado THEN
	LinkDelta.Others := LinkDelta.Others OR 2#100;
ELSE
	LinkDelta.Others := LinkDelta.Others AND 2#011;
END_IF
END_ACTION

ACTION Status:


motor.En.xEmergenciaOK := motor.En.xEmergenciaOK OR NOT LinkDelta.ErrorCode = 76;

motor.En.xTemInversor := TRUE;
tonOnline(IN:= LinkDelta.state <> 0, PT:= T#500MS, Q=> , ET=> );
motor.En.xInversorOnline := NOT tonOnline.q;

tonParaDriverPraTrocarDeReferencia(IN:= NOT motor.En.xInversorOnline, PT:= T#500MS, Q=> , ET=> );
IF  NOT motor.En.xInversorOnline AND NOT tonParaDriverPraTrocarDeReferencia.q THEN
	motor.Sa.xCmdFwd := FALSE;
END_IF

motor.En.xFalhaInversor := LinkDelta.ErrorCode <> 0 AND LinkDelta.ErrorCode <> 49 AND LinkDelta.ErrorCode <> 50 AND LinkDelta.ErrorCode <> 51 AND LinkDelta.ErrorCode <> 76;


rAux := LinkDelta.OutputCurrent;
motor.Sa.rCorrente := rAux/100;

rAux := LinkDelta.OutputFrequence;
motor.Sa.rVelocidadeHz := rAux/100;



IF Motor.Config.xVeloEmMetroPMin THEN	
	rAux := motor.Sa.rVelocidadeHz;
	motor.Sa.rVelocidadeRPM := rAux / (0.016666 * 2);
	rAux										:= (Motor.Sa.rVelocidadeRPM * Motor.Config.rVeloEmMetroPMin_Conversao) / 1800;	
	Motor.Sa.rVeloComissionada				:= rAux;
	Motor.LeiturasInversorIHM.sVelocidadeRPM	:= concat(TO_STRING(F_RetiraCasa(rAux, 2)), ' m/Min');
ELSIF Motor.Config.xVeloEmPorcentagem THEN
	IF Motor.Config.rVeloEmPorcentagem_VeloMax < 0.1 THEN
		Motor.Config.rVeloEmPorcentagem_VeloMax := 1;
	END_IF
	rAux										:= (Motor.Sa.rVelocidadeRPM * 100) / Motor.Config.rVeloEmPorcentagem_VeloMax;
	Motor.Sa.rVeloComissionada				:= rAux;
	Motor.LeiturasInversorIHM.sVelocidadeRPM	:= concat(TO_STRING(F_RetiraCasa(rAux, 2)), ' %');
ELSE
	Motor.Sa.rVeloComissionada				:= Motor.Sa.rVelocidadeRPM;
	Motor.LeiturasInversorIHM.sVelocidadeRPM := concat(TO_STRING(F_RetiraCasa(Motor.Sa.rVelocidadeRPM, 2)), ' RPM');
END_IF


rAux := LinkDelta.DCBusVoltage;
motor.Sa.rVoltagemEntrada := rAux/10 / 1.41;

Motor.LeiturasInversorIHM.sCorrente			:= concat(TO_STRING(F_RetiraCasa(Motor.Sa.rCorrente, 2)), ' A');
Motor.LeiturasInversorIHM.sStatusConexao		:= Motor.Sa.sStatusConexao;
Motor.LeiturasInversorIHM.sTemperaturaInver	:= 'ND';
Motor.LeiturasInversorIHM.sTemperaturaMotor	:= concat(TO_STRING(F_RetiraCasa(Motor.Sa.rTemperaturaMotor, 2)), ' %');
Motor.LeiturasInversorIHM.sTorque				:= concat(TO_STRING(F_RetiraCasa(Motor.Sa.rTorque, 2)), ' %');
Motor.LeiturasInversorIHM.sUltimoErro			:= Motor.Sa.sUltimoErro;
Motor.LeiturasInversorIHM.sVelocidadeHz		:= concat(TO_STRING(F_RetiraCasa(Motor.Sa.rVelocidadeHZ, 2)), ' Hz');






LinkDelta.Out_Value[18] := REAL_TO_UINT(motor.Config.inversor.ACC);
LinkDelta.Out_Value[19] := REAL_TO_UINT(motor.Config.inversor.DEC);
LinkDelta.Out_Value[20] := REAL_TO_UINT(motor.Config.inversor.TFR);


motor.Sa.sStatusConexao := 'Offline';
IF motor.En.xInversorOnline THEN
	motor.Sa.sStatusConexao := 'Online';
	IF motor.En.xFalhaInversor THEN
		motor.Sa.sStatusConexao := 'Falha';	
	END_IF
END_IF



i1ParteStatus := LinkDelta.IN_Value[2] AND 2#0000000000000011;
i2ParteStatus := LinkDelta.IN_Value[2] AND 2#0000000000011000;

(*
CASE i1ParteStatus OF
	0 : motor.Sa.sStatusConexao := 'Parado';
	2 : motor.Sa.sStatusConexao := 'Desligando';
	3 : motor.Sa.sStatusConexao := 'Esperando Comando';
	4 : motor.Sa.sStatusConexao := 'Rodando';
END_CASE

IF i1ParteStatus = 4 THEN
	CASE i2ParteStatus OF
		0  : motor.Sa.sStatusConexao := CONCAT(motor.Sa.sStatusConexao,': frente');
		4  : motor.Sa.sStatusConexao := CONCAT(motor.Sa.sStatusConexao,': Indo para reverso');
		8  : motor.Sa.sStatusConexao := CONCAT(motor.Sa.sStatusConexao,': Indo para frente');
		12 : motor.Sa.sStatusConexao := CONCAT(motor.Sa.sStatusConexao,': Reverso');
	END_CASE
END_IF
*)





CASE LinkDelta.ErrorCode OF
	1 : motor.Sa.sUltimoErro := '[ocA] Sobre-Corrente na aceleração';
	2 : motor.Sa.sUltimoErro := '[ocd] Sobre-Corrente na desaceleração';
	3 : motor.Sa.sUltimoErro := '[ocn] Sobre-Corrente';
	4 : motor.Sa.sUltimoErro := '[GFF] Fuga a terra';
	6 : motor.Sa.sUltimoErro := '[ocS] Sobre-Corrente ao parar';
	7 : motor.Sa.sUltimoErro := '[ouA] Sobre-Corrente na aceleração';
	8 : motor.Sa.sUltimoErro := '[oud] Sobre-Corrente na desaceleração';
	9 : motor.Sa.sUltimoErro := '[oun] Sobre-Tensão em operação normal';
	10 : motor.Sa.sUltimoErro := '[ouS] Sobre-Tensão ao parar';
	11 : motor.Sa.sUltimoErro := '[LuA] Sub-Tensão na aceleração';
	12 : motor.Sa.sUltimoErro := '[Lud] Sub-Tensão na desaceleração';
	13 : motor.Sa.sUltimoErro := '[Lun] Sub-Tensão em operação normal';
	14 : motor.Sa.sUltimoErro := '[Lus] Sub-Tensão ao parar';
	15 : motor.Sa.sUltimoErro := '[orP] Perda de fase';
	16 : motor.Sa.sUltimoErro := '[oHI] IGBT Sobreaquecendo';
	18 : motor.Sa.sUltimoErro := '[THIo] Falha na detecção da temperatura do IGBT';
	21 : motor.Sa.sUltimoErro := '[ol] Sobre Carga';
	22 : motor.Sa.sUltimoErro := '[EoL1] Electronic thermal relay 1 protection';
	23 : motor.Sa.sUltimoErro := '[EoL2] Electronic thermal relay 2 protection';
	24 : motor.Sa.sUltimoErro := '[oh3] Motor Sobreaquecendo';
	26 : motor.Sa.sUltimoErro := '[ot1] Sobre torque 1';
	27 : motor.Sa.sUltimoErro := '[ot2] Sobre torque 2';
	28 : motor.Sa.sUltimoErro := '[uC] Sub-Corrente';
	31 : motor.Sa.sUltimoErro := '[cF2] EEPROM read error';
	33 : motor.Sa.sUltimoErro := '[cd1] Erro na fase U';
	34 : motor.Sa.sUltimoErro := '[cd2] Erro na fase V';
	35 : motor.Sa.sUltimoErro := '[cd3] Erro na fase W';
	36 : motor.Sa.sUltimoErro := '[Hd0] cc hardware error';
	37 : motor.Sa.sUltimoErro := '[Hd1] oc hardware error';
	40 : motor.Sa.sUltimoErro := '[que] Auto-tuning error';
	41 : motor.Sa.sUltimoErro := '[AFE] PID loss ACI';
	43 : motor.Sa.sUltimoErro := '[PGF2] PG feedback loss';
	44 : motor.Sa.sUltimoErro := '[PGF3] PG feedback stall';
	45 : motor.Sa.sUltimoErro := '[PGF4] PG slip error';
	48 : motor.Sa.sUltimoErro := '[ACE] ACI loss';
	49 : motor.Sa.sUltimoErro := '[EF] Emergencia via software';
	50 : motor.Sa.sUltimoErro := '[EF1] Emergencia';
	51 : motor.Sa.sUltimoErro := '[bb] Bloqueio via software';
	52 : motor.Sa.sUltimoErro := '[Pcod] Password is locked';
	54 : motor.Sa.sUltimoErro := '[CE1] Illegal command ';
	55 : motor.Sa.sUltimoErro := '[CE2] Illegal data address';
	56 : motor.Sa.sUltimoErro := '[CE3] Illegal data value';
	57 : motor.Sa.sUltimoErro := '[CE4] Data is written to read-only address';
	58 : motor.Sa.sUltimoErro := '[CE10] Modbus transmission time-out';
	61 : motor.Sa.sUltimoErro := '[ydc] Y-connection / Δ-connection switch error';
	62 : motor.Sa.sUltimoErro := '[dEb] Deceleration energy backup error';
	63 : motor.Sa.sUltimoErro := '[oSL] Erro de escorregamento';
	72 : motor.Sa.sUltimoErro := '[STL1] Perda STO 1';
	76 : motor.Sa.sUltimoErro := '[STO] Emergencia';
	77 : motor.Sa.sUltimoErro := '[STL2] Perda STO 2';
	78 : motor.Sa.sUltimoErro := '[STL3] Perda STO 3';
	79 : motor.Sa.sUltimoErro := '[Aoc] Sobre-Corrente na fase U antes de partir';
	80 : motor.Sa.sUltimoErro := '[boc] Sobre-Corrente na fase V antes de partir';
	81 : motor.Sa.sUltimoErro := '[coc] Sobre-Corrente na fase W antes de partir';
	82 : motor.Sa.sUltimoErro := '[oPL1] Perda da fase U';
	83 : motor.Sa.sUltimoErro := '[oPL2] Perda da fase V';
	84 : motor.Sa.sUltimoErro := '[oPL3] Perda da fase W';
	87 : motor.Sa.sUltimoErro := '[oL3] Proteção de sobrecarga em baixa frequencia';
	89 : motor.Sa.sUltimoErro := '[roPd] Rotor position detection error';
	101 : motor.Sa.sUltimoErro := '[CGdE] CANopen guarding error';
	102 : motor.Sa.sUltimoErro := '[CHbE] CANopen heartbeat error';
	104 : motor.Sa.sUltimoErro := '[CbFE] CANopen bus off error';
	105 : motor.Sa.sUltimoErro := '[CCdE] CANopen index error';
	106 : motor.Sa.sUltimoErro := '[CAdE] CANopen station address error';
	107 : motor.Sa.sUltimoErro := '[CFrE] CANopen index setting exceed limit';
	111 : motor.Sa.sUltimoErro := '[CctE] InrCOM time-out error';
	121 : motor.Sa.sUltimoErro := '[CP20] Internal communication error';
	123 : motor.Sa.sUltimoErro := '[CP22] Internal communication error';
	124 : motor.Sa.sUltimoErro := '[CP30] Internal communication error';
	126 : motor.Sa.sUltimoErro := '[CP32] Internal communication error';
	127 : motor.Sa.sUltimoErro := '[CP33] Internal communication error';
	128 : motor.Sa.sUltimoErro := '[ot3] Over-torque 3';
	129 : motor.Sa.sUltimoErro := '[ot4] Over-torque 4';
	134 : motor.Sa.sUltimoErro := '[Eol3] Internal communication error';
	135 : motor.Sa.sUltimoErro := '[Eol4] Internal communication error';
	140 : motor.Sa.sUltimoErro := '[hd6] oc hardware error';
	141 : motor.Sa.sUltimoErro := '[b4GFF] GFF occurs before run';
	142 : motor.Sa.sUltimoErro := '[AuE1] Auto-tune error 1';
	143 : motor.Sa.sUltimoErro := '[AuE2] Auto-tune error 2';
	144 : motor.Sa.sUltimoErro := '[AuE3] Auto-tune error 3';

END_CASE
END_ACTION

END_FUNCTION_BLOCK

// POUs/Comunicação/ModbusRTU/FB_ControleSoftRTU_LEGADO
FUNCTION_BLOCK FB_ControleSoftRTU_LEGADO
VAR_IN_OUT
	stMotor : st_Partida;
	MestreModbusRTU	: ModbusRtuMasterV2_KL6x22B;
END_VAR
VAR_INPUT
	iEndereco : INT;
	xComeca : BOOL;
END_VAR
VAR_OUTPUT
	xOcupado : BOOL;
	xTerminei : BOOL;
	UltimoErro : STRING;
	xOnline : BOOL;
	rCorrenteL1 : REAL;
	rCorrenteL2 : REAL;
	rCorrenteL3 : REAL;
END_VAR
VAR
	//1 le cempre
	//2 a 4 le quando ta rodadno
	//4 a 8 le quando pede e escreve quando pede
	// 9 e 10 escreve quando inicia pra ficar o controle esperado 
	Registradores 	: ARRAY[1..3] OF INT := [257,258,259];//[279,257,258,259,19,20,1,3,56,74,75];
	Valores			: ARRAY[1..3] OF UINT;

	xAuxOnline : BOOL;
	rtComeca : R_TRIG;
	state : INT;
	tonOnline : TON;
	xBusy : BOOL;
	rAux : REAL;
	
	LFT : INT;
END_VAR

IF xLicensaValida5154156 THEN
	

	rtComeca(CLK := xComeca, Q =>);
	
	IF rtComeca.q THEN
		xAuxOnline := FALSE;
	END_IF
	
	CASE state OF
	
		0:
			// ele so mexe no mestre caso seja a vez dele
			IF xComeca THEN
				MestreModbusRTU.ReadRegs(Execute := FALSE); //bota em 0 pra reiniciar	
				state := 1;
			END_IF
	
		1: //Le registradores
			MestreModbusRTU.ReadRegs
				(
					UnitID := TO_BYTE(iEndereco),
						Quantity := 3,
						MBAddr := TO_WORD(Registradores[1]),
						cbLength := SIZEOF(Valores),
						pMemoryAddr := ADR(Valores),
						Execute := TRUE,
						Timeout := ,
						Busy => xBusy);
	
			IF NOT xBusy THEN
				MestreModbusRTU.ReadRegs(Execute := FALSE);
				// so fica online se ler tudo e nenhumm der erro
				xAuxOnline := MestreModbusRTU.Error;
				// joga de volta pro 0 pra ver se ele terminou
				state		:= 0;
				xTerminei	:= TRUE;
				xComeca		:= FALSE;
			END_IF
	
	END_CASE
	
	tonOnline(IN := NOT xAuxOnline, PT := T#0.5S, Q =>, ET =>);
	xOnline := tonOnline.q;
	
	UltimoErro := MestreModbusRTU.ErrorDiagnostics.LastErrorID;
	
	xOcupado := MestreModbusRTU.BUSY AND xComeca;
	
	rAux	:= TO_INT(Valores[1]);
	rCorrenteL1	:= rAux / 10;
	rAux	:= TO_INT(Valores[2]);
	rCorrenteL2	:= rAux / 10;
	rAux	:= TO_INT(Valores[3]);
	rCorrenteL3	:= rAux / 10;
	
	stMotor.Config.xTemSoft := TRUE;
	stMotor.Sa.rCorrente := (rCorrenteL1+rCorrenteL2+rCorrenteL3)/3;
	stMotor.LeiturasInversorIHM.sCorrente := REAL_TO_STRING(stMotor.Sa.rCorrente);

ELSE
	ValidaLicensa();
END_IF

ACTION Status:



CASE LFT OF
	1 :
		UltimoErro := 'UCF - Subcorrente';
	2 :
		UltimoErro := 'OCF - Sobrecorrente';
	3 :
		UltimoErro := 'PHbd - Fases desbalanceada';
	4 :
		UltimoErro := 'GrdF - Fuga a terra';
	5 :
		UltimoErro := 'OLF - motor sobrecarregado';
	6 :
		UltimoErro := 'OtF - Motor superaquecendo';
	7 :
		UltimoErro := 'OHF - Soft sobreaquecendo';
	8 :
		UltimoErro := 'PIF - Inversão de fase';
	9 :
		UltimoErro := 'PHF - Perda de fase';
	10 :
		UltimoErro := 'USF - subtensão';
	11 :
		UltimoErro := 'OSF - sobretensão';
	12 :
		UltimoErro := 'StF -  Starting time detected fault';
	13 :
		UltimoErro := 'SnbF - Muitas inicializações';
	14 :
		UltimoErro := 'SSCr - conexão errada ou tiristor em curto';
	15 :
		UltimoErro := 'EtF - Falha externa';
	16 :
		UltimoErro := 'InF - Falha interna';
	17 :
		UltimoErro := 'SLF - Modbus erro';
	18 :
		UltimoErro := 'trAp - Codigo trAp';
	19 :
		UltimoErro := 'SCF - Curto-Circuito';
	20 :
		UltimoErro := 'bPF - Contatora de bypass em falha';
	21 :
		UltimoErro := 'CFF - Configuração invalida';
END_CASE
END_ACTION

END_FUNCTION_BLOCK

// POUs/Comunicação/ModbusRTU/FB_ModBusRTU_AC380
//{attribute 'hide_all_locals'}
FUNCTION_BLOCK FB_ModBusRTU_AC380
VAR_IN_OUT
	MestreModbusRTU	: ModbusRtuMasterV2_KL6x22B;
	Motor			: st_Partida;
END_VAR
VAR_INPUT
	xInicia				: BOOL;
END_VAR
VAR_OUTPUT
	//Gerais
	xTerminei				: BOOL;
	UltimoModbusErro		: ST_ModbusErrorDiagnostics;
END_VAR
VAR
	xIniciaInterno				: BOOL;	
	xTerminouLeitura			: BOOL;
	xTerminouEscrita			: BOOL;
	xFalha						: BOOL;
	xInversorOnline				: BOOL;
	xGuardaRegistroErro			: BOOL;
	xRdy						: BOOL;
	xRun						: BOOL;
	xQueimaUmScan				: BOOL;
	ControlWord					: ARRAY[0..15] OF BOOL;

	
	iRegistradorAtual			: INT := 1;
	iEndereco 					: INT;
	i							: INT;
	
	wLeitura					: WORD;
	rVelocidadeAux				: WORD;
	wFalha						: WORD;
	StatusWord					: WORD;
	arLeitura					: ARRAY[1..12] OF WORD;
	arEscrita					: ARRAY[1..3] OF WORD;
	
	RegistradoresLeitura		: ARRAY[1..12] OF INT 	:= [3,100,105,106,109,112,400,410,510,3500,2871,2872];		//Registradores de leitura
	RegistradoresEscrita		: ARRAY[1..3] OF INT 	:= [1,2311,2312];		//Registradores de escrita
	
	stateModbus					: State_Modbus;			//Variável para máquina de estados
	state						: StateWord;
	
	rt							: R_TRIG;				//Inicia vindo de fora
	rtInicia 					: R_TRIG;				//Inicia Leitura/Escrita
	ftInicia					: F_TRIG;				//Para Leitura/Escrita
	
	tTimeout					: TIME := T#1S;			//Tempo de timeout para espera escravo 
	tonTimeOut					: Tc2_Standard.TON;
	
	sStatusConexao				: STRING;
	
	rRampaACCAtual			: REAL;
	rRampaDCCAtual			: REAL;

	
	//Gambiara
	xPodeIrDenovo	: BOOL := TRUE;
END_VAR

IF xLicensaValida5154156 THEN
	rt(CLK := xInicia, Q =>);
	
	IF rt.Q THEN
		xIniciaInterno := TRUE;
	END_IF
	
	
	rtInicia(CLK := xIniciaInterno, Q =>);
	ftInicia(CLK := xIniciaInterno, Q =>);
	
	IF rtInicia.Q THEN
		iRegistradorAtual	:= 1;
		xTerminei			:= FALSE;
		
		//Quando inicia a leitura, não terminou de ler nenhum
		xTerminouLeitura	:= FALSE;
		xTerminouEscrita	:= FALSE;
		
		stateModbus := State_Modbus.Inicia;
		
		iRegistradorAtual := 1;
	END_IF
	
	IF ftInicia.Q  THEN
		xIniciaInterno := FALSE;
		xInicia			:= FALSE;
		iRegistradorAtual := 1;
		xTerminei := TRUE;
		stateModbus := State_Modbus.Inicia;
		MestreModbusRTU.ReadRegs(Execute := FALSE);
		MestreModbusRTU.WriteRegs(Execute := FALSE);
	END_IF
	
	EspelhoEntradas();
	
	Leitura();
	
	Estados();
	
	ExecutaEstados();
	
	Status();
	
	EspelhoSaidas();
	
	Escrita();
	
	tonTimeOut(IN:= MestreModbusRTU.BUSY, PT:= T#10S, Q=> , ET=> );
	
	IF tonTimeOut.Q THEN
		xIniciaInterno := FALSE;
		xInicia := FALSE;
		xInversorOnline := FALSE;
	END_IF
ELSE
	ValidaLicensa();
END_IF

ACTION Escrita:
CASE stateModbus OF
	
	State_Modbus.Inicia:
		IF xIniciaInterno THEN
			MestreModbusRTU.ReadRegs(Execute := FALSE);
			MestreModbusRTU.WriteRegs(Execute := FALSE);

			IF NOT xTerminouLeitura THEN
				stateModbus := State_Modbus.Leitura;
			ELSE
				IF NOT xTerminouEscrita THEN
						stateModbus := State_Modbus.Escrita;
				END_IF
			END_IF;

			IF xTerminouLeitura AND xTerminouEscrita THEN
				xIniciaInterno := FALSE;
				xTerminei := TRUE;
			END_IF
		END_IF
			
	State_Modbus.Escrita:
	
		MestreModbusRTU.WriteRegs(
			UnitID      := TO_BYTE(iEndereco),                 					// Endereço do equipamento escravo na rede Modbus
			Quantity    := 1,                									// Quantidade de WORDs a serem lidas
			MBAddr      := TO_WORD(RegistradoresEscrita[iRegistradorAtual]),	// Endereço Modbus. Onde 0 = Holding Register 40001
			cbLength    := SIZEOF(arEscrita[iRegistradorAtual]), 				// Quantidade de bytes a serem lidos
			pMemoryAddr := ADR(arEscrita[iRegistradorAtual]),					// Ponteiro para o array que receberá os dados lidos
			Execute     := TRUE,              									// Comando para executar o comando    
			Timeout     := tTimeout               								// Tempo de espera da resposta do escravo
		);
		

		IF NOT MestreModbusRTU.BUSY THEN
			IF MestreModbusRTU.Error THEN
				//Se deu erro cai fora
						xTerminouLeitura	:= TRUE;
						xTerminouEscrita	:= TRUE;
						
						stateModbus := State_Modbus.Inicia;
						xIniciaInterno := FALSE;
						
						xGuardaRegistroErro := TRUE;
						
			ELSE
				
				MestreModbusRTU.WriteRegs(Execute := FALSE);
	
				stateModbus := State_Modbus.Inicia;		
				
				iRegistradorAtual := iRegistradorAtual + 1;	
				
				IF iRegistradorAtual > 3 THEN
					stateModbus := State_Modbus.Inicia;
					iRegistradorAtual := 1;
					xTerminouEscrita	:= TRUE;
					
					xGuardaRegistroErro := FALSE;
				END_IF
				
			END_IF
		END_IF 
END_CASE
END_ACTION

ACTION EspelhoEntradas:


arEscrita[1]	:= INT_TO_WORD(Motor.Sa.iVelocidade*10);
arEscrita[2]	:= REAL_TO_WORD(Motor.Config.inversor.ACC*10);
arEscrita[3]	:= REAL_TO_WORD(Motor.Config.inversor.DEC*10);
//arEscrita[4]	:= REAL_TO_WORD(Motor.Config.inversor.ACC*10);
//arEscrita[5]	:= REAL_TO_WORD(Motor.Config.inversor.DEC*10);
iEndereco		:= Motor.En.i;
END_ACTION

ACTION EspelhoSaidas:
IF xTerminouLeitura AND xTerminouEscrita THEN
	Motor.Sa.rVelocidadeRPM		:= WORD_TO_REAL(arLeitura[2])/10;
	Motor.Sa.rVelocidadeHz		:= WORD_TO_REAL(arLeitura[3])/100;
	Motor.Sa.rCorrente			:= WORD_TO_REAL(arLeitura[4])/100;
	Motor.Sa.rTorque			:= WORD_TO_REAL(arLeitura[5])/100;
	Motor.Sa.rVoltagemEntrada	:= WORD_TO_REAL(arLeitura[6]);	//Na verdade, aqui é de saída meu jovem.
	Motor.Sa.rTemperaturaMotor	:= WORD_TO_REAL(arLeitura[9]);
	Motor.Sa.rTemperaturaInver	:= WORD_TO_REAL(arLeitura[10]);
	rRampaACCAtual				:= WORD_TO_REAL(arLeitura[11])/10;
	rRampaDCCAtual				:= WORD_TO_REAL(arLeitura[12])/10;
	Motor.En.xFalhaInversor		:= xFalha;
	Motor.Sa.sStatusConexao		:= sStatusConexao;
	Motor.En.xTemInversor 		:= TRUE;
	Motor.En.xInversorOnline 	:= xInversorOnline;
	UltimoModbusErro			:= MestreModbusRTU.ErrorDiagnostics;
	
	IF NOT xInversorOnline THEN
		Motor.Sa.rVelocidadeRPM := 0;
		Motor.Sa.rVelocidadeHz := 0;
		Motor.Sa.rCorrente := 0;
		Motor.Sa.rTorque := 0;
		Motor.Sa.rVoltagemEntrada :=0;
		Motor.Sa.rTemperaturaMotor := 0;
		Motor.Sa.rTemperaturaInver := 0;
		rRampaACCAtual := 0;
		rRampaDCCAtual := 0;
	END_IF
	
	CASE arLeitura[8] OF
		16#0:
			Motor.Sa.sUltimoErro := 'Inversor Offline';
		16#1080:
			Motor.Sa.sUltimoErro := 'Tempo Limite Backup/Restauração';
		16#1081:
			Motor.Sa.sUltimoErro := 'Falha na classificação do ID';
		16#2281:
			Motor.Sa.sUltimoErro := 'Calibração';
		16#2310:
			Motor.Sa.sUltimoErro := 'Sobrecorrente';
		16#2330:
			Motor.Sa.sUltimoErro := 'Fuga à Terra';
		16#2340:
			Motor.Sa.sUltimoErro := 'Curto-Circuito na Saída';
		16#2381:
			Motor.Sa.sUltimoErro := 'Sobrecarga no IGBT';
		16#3130:
			Motor.Sa.sUltimoErro := 'Falta de Fase na Entrada';
		16#3181:
			Motor.Sa.sUltimoErro := 'Cross Connection';
		16#3210:
			Motor.Sa.sUltimoErro := 'Sobretensão CC no Circuito intermediário';
		16#3220:
			Motor.Sa.sUltimoErro := 'Subtensão CC no Circuito intermediário';
		16#3381:
			Motor.Sa.sUltimoErro := 'Falta de Fase na Saída';
		16#4110:
			Motor.Sa.sUltimoErro := 'Temperatura alta na placa de controle';
		16#4210:
			Motor.Sa.sUltimoErro := 'Sobretemperatura estimada no IGBT';
		16#4290:
			Motor.Sa.sUltimoErro := 'Temperatura alta no módulo do inversor';
		16#42F1:
			Motor.Sa.sUltimoErro := 'Sobretemperatura no IGBT';
		16#4310:
			Motor.Sa.sUltimoErro := 'Temperatura alta no módulo de potência';
		16#4380:
			Motor.Sa.sUltimoErro := 'Diferença de temperatura IGBT';
		16#4981:
			Motor.Sa.sUltimoErro := 'Falha - Temperatura externa 1';
		16#4982:
			Motor.Sa.sUltimoErro := 'Falha - Temperatura externa 2';
		16#5090:
			Motor.Sa.sUltimoErro := 'Falha no Hardware STO';
		16#5091:
			Motor.Sa.sUltimoErro := 'STO - Safe Torque OFF';
		16#5092:
			Motor.Sa.sUltimoErro := 'Erro Lógico PU';
		16#5093:
			Motor.Sa.sUltimoErro := 'Hardware incompatível com Firmware';
		16#5094:
			Motor.Sa.sUltimoErro := 'Falha na Medição de Temperatura interna';
		16#50A0:
			Motor.Sa.sUltimoErro := 'Ventilador de Refrigeração em Falha';
		16#5681:
			Motor.Sa.sUltimoErro := 'Falha na comunicação PU';
		16#5682:
			Motor.Sa.sUltimoErro := 'Unidade de Potência Perdida';
		16#5690:
			Motor.Sa.sUltimoErro := 'Falha na Comunicação Interna';
		16#5691:
			Motor.Sa.sUltimoErro := 'Falha no Circuito de Medição';
		16#5692:
			Motor.Sa.sUltimoErro := 'Falha de Alimentação na Unidade de Potência';
		16#5693:
			Motor.Sa.sUltimoErro := 'Falha no Circuito de Medição';
		16#5696:
			Motor.Sa.sUltimoErro := 'Feedback dos Estados das Fases Incorreto';
		16#5697:
			Motor.Sa.sUltimoErro := 'Sem sinal de Feedback das Fases';
		16#6181:
			Motor.Sa.sUltimoErro := 'Versão da FPGA incompatível com o Firmware';
		16#6306:
			Motor.Sa.sUltimoErro := 'Sem sinal de Feedback das Fases';
		16#6481:
			Motor.Sa.sUltimoErro := 'Falha Interna';
		16#6487:
			Motor.Sa.sUltimoErro := 'Falha Interna';
		16#64A1:
			Motor.Sa.sUltimoErro := 'Erro de Leitura de Arquivo';
		16#64A6:
			Motor.Sa.sUltimoErro := 'Falha no programa adaptativo';
		16#64B2:
			Motor.Sa.sUltimoErro := 'Falha no conjunto de parâmetros utilizados';
		16#64E1:
			Motor.Sa.sUltimoErro := 'Erro de Sistema Operacional';
		16#6581:
			Motor.Sa.sUltimoErro := 'Falha ao salvar/carregar parâmetro';
		16#65A1:
			Motor.Sa.sUltimoErro := 'Informação requerida pelo PLC não disponpivel';
		16#6681:
			Motor.Sa.sUltimoErro := 'Perda comunicação EFB(FieldBus Integrado)';
		16#6682:
			Motor.Sa.sUltimoErro := 'Falha ao ler o arquivo EFB(FieldBus Integrado)';
		16#6683:
			Motor.Sa.sUltimoErro := 'Parâmetro EFB(FieldBus Integrado) inválido';
		16#6684:
			Motor.Sa.sUltimoErro := 'Falha ao carregar o firmware EFB(FieldBus Integrado)';
		16#6685:
			Motor.Sa.sUltimoErro := 'Falha reservada EFB(FieldBus Integrado) 1';
		16#6686:
			Motor.Sa.sUltimoErro := 'Falha reservada EFB(FieldBus Integrado) 2';
		16#6882:
			Motor.Sa.sUltimoErro := 'Falha Interna';
		16#6885:
			Motor.Sa.sUltimoErro := 'Falha Interna';
		16#7081:
			Motor.Sa.sUltimoErro := 'Perda do Painel de Controle';
		16#7082:
			Motor.Sa.sUltimoErro := 'Perda de Comunicação do Módulo I/O';
		16#7086:
			Motor.Sa.sUltimoErro := 'Sobretensão no Módulo I/O';
		16#71A2:
			Motor.Sa.sUltimoErro := 'Falha de Controle do Freio Meânico (Fechamento)';
		16#71A3:
			Motor.Sa.sUltimoErro := 'Falha de Controle do Freio Meânico (Abertura)';
		16#71A5:
			Motor.Sa.sUltimoErro := 'Freio Mecânico Travado';
		16#7121:
			Motor.Sa.sUltimoErro := 'Motor bloqueado: Carga Excessiva ou Energia Insuficiente';
		16#7181:
			Motor.Sa.sUltimoErro := 'Problema na Resistência de Frenagem';
		16#7183:
			Motor.Sa.sUltimoErro := 'Temperatura Alta na Resistência de Frenagem';
		16#7184:
			Motor.Sa.sUltimoErro := 'Curto-Circuito na Resistência de Frenagem';
		16#7191:
			Motor.Sa.sUltimoErro := 'Curto-Circuito no Chopper IGBT';
		16#7192:
			Motor.Sa.sUltimoErro := 'Temperatura Alta no Chopper IGBT';
		16#7301:
			Motor.Sa.sUltimoErro := 'Sem Feedback de Velocidade do Motor';
		16#7310:
			Motor.Sa.sUltimoErro := 'Sobrevelocidade';
		16#7381:
			Motor.Sa.sUltimoErro := 'Falha no Feedback do Encoder';
		16#73F0:
			Motor.Sa.sUltimoErro := 'Sobrefrequência';
		16#73B0:
			Motor.Sa.sUltimoErro := 'Falha na Parada de Emergência';
		16#7510:
			Motor.Sa.sUltimoErro := 'Perda de comunicação FBA A';
		16#8001:
			Motor.Sa.sUltimoErro := 'Falha de subcarga (Abaixo)';
		16#8002:
			Motor.Sa.sUltimoErro := 'Falha de subcarga (Acima)';
		16#80A0:
			Motor.Sa.sUltimoErro := 'Sinal Analógico Fora dos Limites';
		16#80B0:
			Motor.Sa.sUltimoErro := 'Falha Supervisão de Sinal 66';
		16#80B1:
			Motor.Sa.sUltimoErro := 'Falha Supervisão de Sinal 66';
		16#80B2:
			Motor.Sa.sUltimoErro := 'Falha Supervisão de Sinal 66';
		16#80B3:
			Motor.Sa.sUltimoErro := 'Falha Supervisão de Sinal 66';
		16#80B4:
			Motor.Sa.sUltimoErro := 'Falha Supervisão de Sinal 66';
		16#80B5:
			Motor.Sa.sUltimoErro := 'Falha Supervisão de Sinal 66';
		16#9081:
			Motor.Sa.sUltimoErro := 'Falha Dispotivo Externo 1';
		16#9082:
			Motor.Sa.sUltimoErro := 'Falha Dispotivo Externo 2';
		16#9083:
			Motor.Sa.sUltimoErro := 'Falha Dispotivo Externo 3';
		16#9084:
			Motor.Sa.sUltimoErro := 'Falha Dispotivo Externo 4';
		16#9085:
			Motor.Sa.sUltimoErro := 'Falha Dispotivo Externo 5';
		16#FA81:
			Motor.Sa.sUltimoErro := 'STO (Safe Torque OFF) 1 rompido';
		16#FA82:
			Motor.Sa.sUltimoErro := 'STO (Safe Torque OFF) 1 rompido';
		16#FF61:
			Motor.Sa.sUltimoErro := 'ID Run';
		16#FF81:
			Motor.Sa.sUltimoErro := 'Falha forçada FBA';
		16#FF8E:
			Motor.Sa.sUltimoErro := 'Falha forçada FBB';
		16#D100:
			Motor.Sa.sUltimoErro := 'Inversor não Consegiu Fornecer Torque Suficiente';
		16#D101:
			Motor.Sa.sUltimoErro := 'Escorregamento do Freio';
		16#D102:
			Motor.Sa.sUltimoErro := 'Velocidade abaixo do limite de segurança';
		16#D105:
			Motor.Sa.sUltimoErro := 'Velocidade do motor Excedeu o Desvio De Estado Estacionário';
		16#D108:
			Motor.Sa.sUltimoErro := 'Comando de limite de parada Frente e Ré Ativos Simultaneamente';
	END_CASE
END_IF
END_ACTION

ACTION Estados:
StatusWord.0;
StatusWord.1;
StatusWord.2;
StatusWord.3;
StatusWord.4;
StatusWord.5;
StatusWord.6;
StatusWord.7;
StatusWord.8;
StatusWord.9;
StatusWord.10;
StatusWord.11;
StatusWord.12;
StatusWord.13;
StatusWord.14;
StatusWord.15;
(*
//Pronto
IF StatusWord.0 THEN
	xRdy := TRUE;
ELSE
	xRdy := FALSE;
END_IF
*)
//Run
IF StatusWord.0 AND StatusWord.1 AND StatusWord.2 THEN
	xRun := TRUE;
ELSE
	xRun := FALSE;
END_IF

//Falha ou STO
IF StatusWord.3 OR NOT StatusWord.4 OR NOT StatusWord.5 THEN
	xFalha	:= TRUE;
ELSE
	xFalha	:= FALSE;
END_IF
END_ACTION

ACTION ExecutaEstados:

END_ACTION

ACTION Leitura:
CASE stateModbus OF
	
	State_Modbus.Inicia:
		IF xIniciaInterno THEN
			MestreModbusRTU.ReadRegs(Execute := FALSE);
			MestreModbusRTU.WriteSingleRegister(Execute := FALSE);

			//Se não terminou de ler corrente, fica lendo a corrente	
			IF NOT xTerminouLeitura THEN
				stateModbus := State_Modbus.Leitura;
			ELSE
				IF NOT xTerminouEscrita THEN
					stateModbus := State_Modbus.Escrita;
				END_IF
			END_IF;

			IF xTerminouLeitura AND xTerminouEscrita THEN
				xIniciaInterno := FALSE;
				xTerminei := TRUE;
			END_IF
		END_IF
		


	//Leitura
	State_Modbus.Leitura:
		
		MestreModbusRTU.ReadRegs(
			UnitID      := TO_BYTE(iEndereco),                 					// Endereço do equipamento escravo na rede Modbus
			Quantity    := 1,                									// Quantidade de WORDs a serem lidas
			MBAddr      := TO_WORD(RegistradoresLeitura[iRegistradorAtual]),	// Endereço Modbus. Onde 0 = Holding Register 40001
			cbLength    := SIZEOF(arLeitura[iRegistradorAtual]),				// Quantidade de bytes a serem lidos
			pMemoryAddr := ADR(arLeitura[iRegistradorAtual]),					// Ponteiro para o array que receberá os dados lidos
			Execute     := TRUE,              									// Comando para executar o comando    
			Timeout     := tTimeout               								// Tempo de espera da resposta do escravo
		);
	
			IF NOT MestreModbusRTU.BUSY THEN
				IF MestreModbusRTU.Error THEN
					//Se deu erro cai fora
						xTerminouLeitura	:= TRUE;
						xTerminouEscrita	:= TRUE;
						
						stateModbus := State_Modbus.Inicia;
						xIniciaInterno := FALSE;
						
						xGuardaRegistroErro := TRUE;
						
				END_IF
				
				MestreModbusRTU.ReadRegs(Execute := FALSE);
				
				iRegistradorAtual := iRegistradorAtual + 1;					
		
				stateModbus := State_Modbus.Inicia;	

	
				
				IF iRegistradorAtual > 12 THEN
					stateModbus := State_Modbus.Inicia;
					iRegistradorAtual := 1;
					xTerminouLeitura := TRUE;
					
					(*wLeitura := arLeitura[1];
					FOR i := 1 TO 11 DO
						arLeitura[i] := arLeitura[i+1];
					END_FOR
					arLeitura[12] := wLeitura;*)
				
				END_IF
			END_IF 
			
END_CASE

StatusWord		:= arLeitura[1];
wFalha			:= arLeitura[7];
END_ACTION

ACTION Leitura_Escrita:
CASE stateModbus OF
	
	State_Modbus.Inicia:
		IF xIniciaInterno THEN
			MestreModbusRTU.ReadRegs(Execute := FALSE);
			MestreModbusRTU.WriteSingleCoil(Execute := FALSE);

			//Se não terminou de ler corrente, fica lendo a corrente	
			IF NOT xTerminouLeitura THEN
				stateModbus := State_Modbus.Leitura;
			ELSE
				IF NOT xTerminouEscrita THEN
					stateModbus := State_Modbus.Escrita;
				END_IF
			END_IF;

			IF xTerminouLeitura AND xTerminouEscrita THEN
				xIniciaInterno := FALSE;
				xTerminei := TRUE;
			END_IF
		END_IF
		


	//Leitura
	State_Modbus.Leitura:
		
		MestreModbusRTU.ReadRegs(
			UnitID      := TO_BYTE(iEndereco),                 					// Endereço do equipamento escravo na rede Modbus
			Quantity    := 1,                									// Quantidade de WORDs a serem lidas
			MBAddr      := TO_WORD(RegistradoresLeitura[iRegistradorAtual]),	// Endereço Modbus. Onde 0 = Holding Register 40001
			cbLength    := SIZEOF(wLeitura), 									// Quantidade de bytes a serem lidos
			pMemoryAddr := ADR(wLeitura),    									// Ponteiro para o array que receberá os dados lidos
			Execute     := TRUE,              									// Comando para executar o comando    
			Timeout     := tTimeout               								// Tempo de espera da resposta do escravo
		);
	
			IF NOT MestreModbusRTU.BUSY THEN
				IF MestreModbusRTU.Error THEN
					//Se deu erro cai fora
						xTerminouLeitura	:= TRUE;
						xTerminouEscrita	:= TRUE;
						
						stateModbus := State_Modbus.Inicia;
						xIniciaInterno := FALSE;
				END_IF

				MestreModbusRTU.ReadRegs(Execute := FALSE);
				
				arLeitura[iRegistradorAtual] := wLeitura;
			
				iRegistradorAtual := iRegistradorAtual + 1;	
		
				stateModbus := State_Modbus.Inicia;		
				
				IF iRegistradorAtual > 12 THEN
					stateModbus := State_Modbus.Escrita;
					iRegistradorAtual := 1;
					xTerminouLeitura := TRUE;
				END_IF
			END_IF 
			
	State_Modbus.Escrita:
	
		MestreModbusRTU.WriteSingleRegister(
			UnitID      := TO_BYTE(iEndereco),                 					// Endereço do equipamento escravo na rede Modbus
			Quantity    := 1,                									// Quantidade de WORDs a serem lidas
			MBAddr      := TO_WORD(RegistradoresEscrita[iRegistradorAtual]),	// Endereço Modbus. Onde 0 = Holding Register 40001
			cbLength    := SIZEOF(arEscrita[iRegistradorAtual]), 				// Quantidade de bytes a serem lidos
			pMemoryAddr := ADR(arEscrita[iRegistradorAtual]),					// Ponteiro para o array que receberá os dados lidos
			Execute     := TRUE,              									// Comando para executar o comando    
			Timeout     := tTimeout               								// Tempo de espera da resposta do escravo
		);

		IF NOT MestreModbusRTU.BUSY THEN
			IF MestreModbusRTU.Error THEN
				//Se deu erro cai fora
						xTerminouLeitura	:= TRUE;
						xTerminouEscrita	:= TRUE;
						
						stateModbus := State_Modbus.Inicia;
						xIniciaInterno := FALSE;
			END_IF
			
			MestreModbusRTU.WriteSingleRegister(Execute := FALSE);
	
			stateModbus := State_Modbus.Inicia;		
			
			iRegistradorAtual := iRegistradorAtual + 1;	
			
			IF iRegistradorAtual > 3 THEN
				stateModbus := State_Modbus.Inicia;
				iRegistradorAtual := 1;
				xTerminouEscrita	:= TRUE;
			END_IF

		END_IF 
END_CASE
END_ACTION

ACTION Status:
xInversorOnline := TRUE;

IF xFalha THEN
	CASE wFalha OF
		16#0:
			sStatusConexao := 'Inversor Offline';
			xInversorOnline := FALSE;
		16#1080:
			sStatusConexao := 'Tempo Limite Backup/Restauração';
		16#1081:
			sStatusConexao := 'Falha na classificação do ID';
		16#2281:
			sStatusConexao := 'Calibração';
		16#2310:
			sStatusConexao := 'Sobrecorrente';
		16#2330:
			sStatusConexao := 'Fuga à Terra';
		16#2340:
			sStatusConexao := 'Curto-Circuito na Saída';
		16#2381:
			sStatusConexao := 'Sobrecarga no IGBT';
		16#3130:
			sStatusConexao := 'Falta de Fase na Entrada';
		16#3181:
			sStatusConexao := 'Cross Connection';
		16#3210:
			sStatusConexao := 'Sobretensão CC no Circuito intermediário';
		16#3220:
			sStatusConexao := 'Subtensão CC no Circuito intermediário';
		16#3381:
			sStatusConexao := 'Falta de Fase na Saída';
		16#4110:
			sStatusConexao := 'Temperatura alta na placa de controle';
		16#4210:
			sStatusConexao := 'Sobretemperatura estimada no IGBT';
		16#4290:
			sStatusConexao := 'Temperatura alta no módulo do inversor';
		16#42F1:
			sStatusConexao := 'Sobretemperatura no IGBT';
		16#4310:
			sStatusConexao := 'Temperatura alta no módulo de potência';
		16#4380:
			sStatusConexao := 'Diferença de temperatura IGBT';
		16#4981:
			sStatusConexao := 'Falha - Temperatura externa 1';
		16#4982:
			sStatusConexao := 'Falha - Temperatura externa 2';
		16#5090:
			sStatusConexao := 'Falha no Hardware STO';
		16#5091:
			sStatusConexao := 'STO - Safe Torque OFF';
		16#5092:
			sStatusConexao := 'Erro Lógico PU';
		16#5093:
			sStatusConexao := 'Hardware incompatível com Firmware';
		16#5094:
			sStatusConexao := 'Falha na Medição de Temperatura interna';
		16#50A0:
			sStatusConexao := 'Ventilador de Refrigeração em Falha';
		16#5681:
			sStatusConexao := 'Falha na comunicação PU';
		16#5682:
			sStatusConexao := 'Unidade de Potência Perdida';
		16#5690:
			sStatusConexao := 'Falha na Comunicação Interna';
		16#5691:
			sStatusConexao := 'Falha no Circuito de Medição';
		16#5692:
			sStatusConexao := 'Falha de Alimentação na Unidade de Potência';
		16#5693:
			sStatusConexao := 'Falha no Circuito de Medição';
		16#5696:
			sStatusConexao := 'Feedback dos Estados das Fases Incorreto';
		16#5697:
			sStatusConexao := 'Sem sinal de Feedback das Fases';
		16#6181:
			sStatusConexao := 'Versão da FPGA incompatível com o Firmware';
		16#6306:
			sStatusConexao := 'Sem sinal de Feedback das Fases';
		16#6481:
			sStatusConexao := 'Falha Interna';
		16#6487:
			sStatusConexao := 'Falha Interna';
		16#64A1:
			sStatusConexao := 'Erro de Leitura de Arquivo';
		16#64A6:
			sStatusConexao := 'Falha no programa adaptativo';
		16#64B2:
			sStatusConexao := 'Falha no conjunto de parâmetros utilizados';
		16#64E1:
			sStatusConexao := 'Erro de Sistema Operacional';
		16#6581:
			sStatusConexao := 'Falha ao salvar/carregar parâmetro';
		16#65A1:
			sStatusConexao := 'Informação requerida pelo PLC não disponpivel';
		16#6681:
			sStatusConexao := 'Perda comunicação EFB(FieldBus Integrado)';
		16#6682:
			sStatusConexao := 'Falha ao ler o arquivo EFB(FieldBus Integrado)';
		16#6683:
			sStatusConexao := 'Parâmetro EFB(FieldBus Integrado) inválido';
		16#6684:
			sStatusConexao := 'Falha ao carregar o firmware EFB(FieldBus Integrado)';
		16#6685:
			sStatusConexao := 'Falha reservada EFB(FieldBus Integrado) 1';
		16#6686:
			sStatusConexao := 'Falha reservada EFB(FieldBus Integrado) 2';
		16#6882:
			sStatusConexao := 'Falha Interna';
		16#6885:
			sStatusConexao := 'Falha Interna';
		16#7081:
			sStatusConexao := 'Perda do Painel de Controle';
		16#7082:
			sStatusConexao := 'Perda de Comunicação do Módulo I/O';
		16#7086:
			sStatusConexao := 'Sobretensão no Módulo I/O';
		16#71A2:
			sStatusConexao := 'Falha de Controle do Freio Meânico (Fechamento)';
		16#71A3:
			sStatusConexao := 'Falha de Controle do Freio Meânico (Abertura)';
		16#71A5:
			sStatusConexao := 'Freio Mecânico Travado';
		16#7121:
			sStatusConexao := 'Motor bloqueado: Carga Excessiva ou Energia Insuficiente';
		16#7181:
			sStatusConexao := 'Problema na Resistência de Frenagem';
		16#7183:
			sStatusConexao := 'Temperatura Alta na Resistência de Frenagem';
		16#7184:
			sStatusConexao := 'Curto-Circuito na Resistência de Frenagem';
		16#7191:
			sStatusConexao := 'Curto-Circuito no Chopper IGBT';
		16#7192:
			sStatusConexao := 'Temperatura Alta no Chopper IGBT';
		16#7301:
			sStatusConexao := 'Sem Feedback de Velocidade do Motor';
		16#7310:
			sStatusConexao := 'Sobrevelocidade';
		16#7381:
			sStatusConexao := 'Falha no Feedback do Encoder';
		16#73F0:
			sStatusConexao := 'Sobrefrequência';
		16#73B0:
			sStatusConexao := 'Falha na Parada de Emergência';
		16#7510:
			sStatusConexao := 'Perda de comunicação FBA A';
		16#8001:
			sStatusConexao := 'Falha de subcarga (Abaixo)';
		16#8002:
			sStatusConexao := 'Falha de subcarga (Acima)';
		16#80A0:
			sStatusConexao := 'Sinal Analógico Fora dos Limites';
		16#80B0:
			sStatusConexao := 'Falha Supervisão de Sinal 66';
		16#80B1:
			sStatusConexao := 'Falha Supervisão de Sinal 66';
		16#80B2:
			sStatusConexao := 'Falha Supervisão de Sinal 66';
		16#80B3:
			sStatusConexao := 'Falha Supervisão de Sinal 66';
		16#80B4:
			sStatusConexao := 'Falha Supervisão de Sinal 66';
		16#80B5:
			sStatusConexao := 'Falha Supervisão de Sinal 66';
		16#9081:
			sStatusConexao := 'Falha Dispotivo Externo 1';
		16#9082:
			sStatusConexao := 'Falha Dispotivo Externo 2';
		16#9083:
			sStatusConexao := 'Falha Dispotivo Externo 3';
		16#9084:
			sStatusConexao := 'Falha Dispotivo Externo 4';
		16#9085:
			sStatusConexao := 'Falha Dispotivo Externo 5';
		16#FA81:
			sStatusConexao := 'STO (Safe Torque OFF) 1 rompido';
		16#FA82:
			sStatusConexao := 'STO (Safe Torque OFF) 1 rompido';
		16#FF61:
			sStatusConexao := 'ID Run';
		16#FF81:
			sStatusConexao := 'Falha forçada FBA';
		16#FF8E:
			sStatusConexao := 'Falha forçada FBB';
		16#D100:
			sStatusConexao := 'Inversor não Consegiu Fornecer Torque Suficiente';
		16#D101:
			sStatusConexao := 'Escorregamento do Freio';
		16#D102:
			sStatusConexao := 'Velocidade abaixo do limite de segurança';
		16#D105:
			sStatusConexao := 'Velocidade do motor Excedeu o Desvio De Estado Estacionário';
		16#D108:
			sStatusConexao := 'Comando de limite de parada Frente e Ré Ativos Simultaneamente';
	END_CASE
ELSE
	IF NOT xRun AND NOT Motor.Sa.xFalha THEN
		sStatusConexao := 'Pronto para Rodar';
	ELSE
		sStatusConexao := 'Rodando';
	END_IF
	
	IF Motor.Sa.xFalha THEN
		sStatusConexao := 'Inversor OK / Falha na Partida';
	END_IF
END_IF

IF xGuardaRegistroErro THEN
	xInversorOnline := FALSE;
END_IF
END_ACTION

END_FUNCTION_BLOCK

// POUs/Comunicação/ModbusRTU/FB_ModBusRTU_ALTISTAR22
{attribute 'hide_all_locals'}
FUNCTION_BLOCK FB_ModBusRTU_ALTISTAR22
VAR_IN_OUT
	MestreModbusRTU	: ModbusRtuMasterV2_KL6x22B;
	Motor			: st_Partida;
END_VAR
VAR_INPUT
	xInicia				: BOOL;
END_VAR
VAR_OUTPUT
	//Gerais
	xTerminei				: BOOL;
	UltimoModbusErro		: ST_ModbusErrorDiagnostics;
END_VAR
VAR
	xIniciaInterno				: BOOL;	
	xTerminouLeitura			: BOOL;
	xTerminouEscrita			: BOOL;
	xSoftOnline					: BOOL;
	xGuardaRegistroErro			: BOOL;
	ControlWord					:  WORD;

	
